LIN {X 0,Y 279.71,Z 650.698,A -85,B 0,C 180,E1 18893.052,E2 18893.052} C_VEL
LIN {X 0,Y 279.473,Z 647.41,A -85,B 0,C 180,E1 18896.902,E2 18896.902} C_VEL
LIN {X 0,Y 279.75,Z 647.577,A -85,B 0,C 180,E1 18903.089,E2 18903.089} C_VEL
LIN {X 0,Y 281.999,Z 655.241,A -85,B 0,C 180,E1 18910.89,E2 18910.89} C_VEL
LIN {X 0,Y 286.328,Z 667.268,A -85,B 0,C 180,E1 18917.884,E2 18917.884} C_VEL
LIN {X 0,Y 291.188,Z 684.37,A -85,B 0,C 180,E1 18924.489,E2 18924.489} C_VEL
LIN {X 0,Y 294.308,Z 701.563,A -85,B 0,C 180,E1 18929.526,E2 18929.526} C_VEL
LIN {X 0,Y 294.245,Z 706.547,A -85,B 0,C 180,E1 18930.593,E2 18930.593} C_VEL
LIN {X 0,Y 277.927,Z 740.652,A -85,B 0,C 180,E1 18934.449,E2 18934.449} C_VEL
LIN {X 0,Y 260.322,Z 771.594,A -85,B 0,C 180,E1 18939.724,E2 18939.724} C_VEL
LIN {X 0,Y 242.682,Z 798.964,A -85,B 0,C 180,E1 18946.842,E2 18946.842} C_VEL
LIN {X 0,Y 228.545,Z 820.039,A -85,B 0,C 180,E1 18955.34,E2 18955.34} C_VEL
LIN {X 0,Y 219.447,Z 834.564,A -85,B 0,C 180,E1 18964.163,E2 18964.163} C_VEL
LIN {X 0,Y 214.489,Z 844.444,A -85,B 0,C 180,E1 18973.653,E2 18973.653} C_VEL
LIN {X 0,Y 212.912,Z 849.596,A -85,B 0,C 180,E1 18982.818,E2 18982.818} C_VEL
LIN {X 0,Y 213.05,Z 850.932,A -85,B 0,C 180,E1 18989.998,E2 18989.998} C_VEL
LIN {X 0,Y 213.023,Z 849.298,A -85,B 0,C 180,E1 18998.143,E2 18998.143} C_VEL
LIN {X 0,Y 215.057,Z 843.186,A -85,B 0,C 180,E1 19007.864,E2 19007.864} C_VEL
LIN {X 0,Y 221.626,Z 830.85,A -85,B 0,C 180,E1 19018.463,E2 19018.463} C_VEL
LIN {X 0,Y 233.239,Z 812.967,A -85,B 0,C 180,E1 19027.923,E2 19027.923} C_VEL
LIN {X 0,Y 248.433,Z 790.316,A -85,B 0,C 180,E1 19035.767,E2 19035.767} C_VEL
LIN {X 0,Y 266.81,Z 760.833,A -85,B 0,C 180,E1 19042.352,E2 19042.352} C_VEL
LIN {X 0,Y 283.537,Z 729.753,A -85,B 0,C 180,E1 19046.951,E2 19046.951} C_VEL
LIN {X 0,Y 294.778,Z 704.676,A -85,B 0,C 180,E1 19049.641,E2 19049.641} C_VEL
LIN {X 0,Y 291.411,Z 685.648,A -85,B 0,C 180,E1 19055.123,E2 19055.123} C_VEL
LIN {X 0,Y 286.674,Z 668.443,A -85,B 0,C 180,E1 19061.593,E2 19061.593} C_VEL
LIN {X 0,Y 282.271,Z 656.335,A -85,B 0,C 180,E1 19068.437,E2 19068.437} C_VEL
LIN {X 0,Y 279.745,Z 647.591,A -85,B 0,C 180,E1 19076.911,E2 19076.911} C_VEL
LIN {X 0,Y 279.623,Z 648.198,A -85,B 0,C 180,E1 19084.646,E2 19084.646} C_VEL
LIN {X 0,Y 282.116,Z 657.702,A -85,B 0,C 180,E1 19093.333,E2 19093.333} C_VEL
LIN {X 0,Y 284.286,Z 663.444,A -85,B 0,C 180,E1 19096.986,E2 19096.986} C_VEL
LIN {X 0,Y 285.392,Z 671.54,A -85,B 0,C 180,E1 19100.105,E2 19100.105} C_VEL
LIN {X 0,Y 286.571,Z 678.848,A -85,B 0,C 180,E1 19102.801,E2 19102.801} C_VEL
LIN {X 0,Y 287.06,Z 679.466,A -85,B 0,C 180,E1 19103.209,E2 19103.209} C_VEL
LIN {X 0,Y 296.62,Z 688.965,A -85,B 0,C 180,E1 19110.583,E2 19110.583} C_VEL
LIN {X 0,Y 304.92,Z 697.051,A -85,B 0,C 180,E1 19117.646,E2 19117.646} C_VEL
LIN {X 0,Y 310.971,Z 702.902,A -85,B 0,C 180,E1 19123.292,E2 19123.292} C_VEL
LIN {X 0,Y 317.433,Z 707.926,A -85,B 0,C 180,E1 19129.521,E2 19129.521} C_VEL
LIN {X 0,Y 322.526,Z 713.626,A -85,B 0,C 180,E1 19135.846,E2 19135.846} C_VEL
LIN {X 0,Y 328,Z 717.173,A -85,B 0,C 180,E1 19142.61,E2 19142.61} C_VEL
LIN {X 0,Y 331.079,Z 721.22,A -85,B 0,C 180,E1 19148.617,E2 19148.617} C_VEL
LIN {X 0,Y 333.856,Z 723.286,A -85,B 0,C 180,E1 19154.266,E2 19154.266} C_VEL
LIN {X 0,Y 336.214,Z 724.311,A -85,B 0,C 180,E1 19160.911,E2 19160.911} C_VEL
LIN {X 0,Y 337.443,Z 724.686,A -85,B 0,C 180,E1 19167.438,E2 19167.438} C_VEL
LIN {X 0,Y 337.436,Z 724.65,A -85,B 0,C 180,E1 19172.564,E2 19172.564} C_VEL
LIN {X 0,Y 336.199,Z 724.407,A -85,B 0,C 180,E1 19179.073,E2 19179.073} C_VEL
LIN {X 0,Y 333.833,Z 723.34,A -85,B 0,C 180,E1 19185.738,E2 19185.738} C_VEL
LIN {X 0,Y 331.067,Z 721.202,A -85,B 0,C 180,E1 19191.387,E2 19191.387} C_VEL
LIN {X 0,Y 327.984,Z 717.14,A -85,B 0,C 180,E1 19197.394,E2 19197.394} C_VEL
LIN {X 0,Y 322.464,Z 713.679,A -85,B 0,C 180,E1 19204.165,E2 19204.165} C_VEL
LIN {X 0,Y 317.373,Z 708.007,A -85,B 0,C 180,E1 19210.466,E2 19210.466} C_VEL
LIN {X 0,Y 310.615,Z 702.32,A -85,B 0,C 180,E1 19217.142,E2 19217.142} C_VEL
LIN {X 0,Y 304.91,Z 697.046,A -85,B 0,C 180,E1 19222.36,E2 19222.36} C_VEL
LIN {X 0,Y 296.59,Z 689.035,A -85,B 0,C 180,E1 19229.414,E2 19229.414} C_VEL
LIN {X 0,Y 287.064,Z 679.509,A -85,B 0,C 180,E1 19236.778,E2 19236.778} C_VEL
LIN {X 0,Y 277.455,Z 660.263,A -85,B 0,C 180,E1 19250.606,E2 19250.606} C_VEL
LIN {X 0,Y 276.701,Z 654.851,A -85,B 0,C 180,E1 19256.871,E2 19256.871} C_VEL
LIN {X 0,Y 276.958,Z 655.076,A -85,B 0,C 180,E1 19263.12,E2 19263.12} C_VEL
LIN {X 0,Y 279.068,Z 662.883,A -85,B 0,C 180,E1 19271.006,E2 19271.006} C_VEL
LIN {X 0,Y 282.954,Z 675.27,A -85,B 0,C 180,E1 19278.105,E2 19278.105} C_VEL
LIN {X 0,Y 286.969,Z 691.731,A -85,B 0,C 180,E1 19284.459,E2 19284.459} C_VEL
LIN {X 0,Y 289.199,Z 707.601,A -85,B 0,C 180,E1 19289.177,E2 19289.177} C_VEL
LIN {X 0,Y 285.282,Z 717.102,A -85,B 0,C 180,E1 19290.276,E2 19290.276} C_VEL
LIN {X 0,Y 268.829,Z 748.728,A -85,B 0,C 180,E1 19294.252,E2 19294.252} C_VEL
LIN {X 0,Y 249.642,Z 780.01,A -85,B 0,C 180,E1 19300.256,E2 19300.256} C_VEL
LIN {X 0,Y 232.045,Z 805.376,A -85,B 0,C 180,E1 19307.849,E2 19307.849} C_VEL
LIN {X 0,Y 218.763,Z 824.231,A -85,B 0,C 180,E1 19316.505,E2 19316.505} C_VEL
LIN {X 0,Y 209.653,Z 838.359,A -85,B 0,C 180,E1 19326.678,E2 19326.678} C_VEL
LIN {X 0,Y 205.697,Z 847.028,A -85,B 0,C 180,E1 19337.284,E2 19337.284} C_VEL
LIN {X 0,Y 204.932,Z 850.268,A -85,B 0,C 180,E1 19345.775,E2 19345.775} C_VEL
LIN {X 0,Y 205.148,Z 850.687,A -85,B 0,C 180,E1 19349.998,E2 19349.998} C_VEL
LIN {X 0,Y 205.128,Z 849.05,A -85,B 0,C 180,E1 19358.459,E2 19358.459} C_VEL
LIN {X 0,Y 207.597,Z 842.427,A -85,B 0,C 180,E1 19369.114,E2 19369.114} C_VEL
LIN {X 0,Y 215.505,Z 829.154,A -85,B 0,C 180,E1 19380.506,E2 19380.506} C_VEL
LIN {X 0,Y 229.199,Z 809.498,A -85,B 0,C 180,E1 19390.551,E2 19390.551} C_VEL
LIN {X 0,Y 245.466,Z 786.097,A -85,B 0,C 180,E1 19398.19,E2 19398.19} C_VEL
LIN {X 0,Y 262.927,Z 758.998,A -85,B 0,C 180,E1 19404.049,E2 19404.049} C_VEL
LIN {X 0,Y 280.537,Z 726.908,A -85,B 0,C 180,E1 19408.637,E2 19408.637} C_VEL
LIN {X 0,Y 289.269,Z 707.475,A -85,B 0,C 180,E1 19410.83,E2 19410.83} C_VEL
LIN {X 0,Y 286.395,Z 689.538,A -85,B 0,C 180,E1 19416.316,E2 19416.316} C_VEL
LIN {X 0,Y 282.277,Z 673.086,A -85,B 0,C 180,E1 19422.932,E2 19422.932} C_VEL
LIN {X 0,Y 278.966,Z 662.903,A -85,B 0,C 180,E1 19429.087,E2 19429.087} C_VEL
LIN {X 0,Y 276.948,Z 655.104,A -85,B 0,C 180,E1 19436.88,E2 19436.88} C_VEL
LIN {X 0,Y 276.7,Z 654.855,A -85,B 0,C 180,E1 19443.129,E2 19443.129} C_VEL
LIN {X 0,Y 278.24,Z 663.042,A -85,B 0,C 180,E1 19451.738,E2 19451.738} C_VEL
LIN {X 0,Y 287.06,Z 679.466,A -85,B 0,C 180,E1 19463.209,E2 19463.209} C_VEL
LIN {X 0,Y 289.006,Z 684.819,A -85,B 0,C 180,E1 19465.563,E2 19465.563} C_VEL
LIN {X 0,Y 290.681,Z 693.974,A -85,B 0,C 180,E1 19469.032,E2 19469.032} C_VEL
LIN {X 0,Y 291.141,Z 694.55,A -85,B 0,C 180,E1 19469.439,E2 19469.439} C_VEL
LIN {X 0,Y 298.491,Z 701.701,A -85,B 0,C 180,E1 19475.552,E2 19475.552} C_VEL
LIN {X 0,Y 306.17,Z 708.716,A -85,B 0,C 180,E1 19482.33,E2 19482.33} C_VEL
LIN {X 0,Y 312.801,Z 714.233,A -85,B 0,C 180,E1 19488.698,E2 19488.698} C_VEL
LIN {X 0,Y 318.348,Z 720.203,A -85,B 0,C 180,E1 19495.334,E2 19495.334} C_VEL
LIN {X 0,Y 324.017,Z 723.954,A -85,B 0,C 180,E1 19502.245,E2 19502.245} C_VEL
LIN {X 0,Y 327.263,Z 728.048,A -85,B 0,C 180,E1 19508.355,E2 19508.355} C_VEL
LIN {X 0,Y 330.039,Z 730.171,A -85,B 0,C 180,E1 19514.079,E2 19514.079} C_VEL
LIN {X 0,Y 332.214,Z 731.196,A -85,B 0,C 180,E1 19519.533,E2 19519.533} C_VEL
LIN {X 0,Y 333.565,Z 731.668,A -85,B 0,C 180,E1 19524.81,E2 19524.81} C_VEL
LIN {X 0,Y 333.984,Z 731.746,A -85,B 0,C 180,E1 19530.001,E2 19530.001} C_VEL
LIN {X 0,Y 333.504,Z 731.607,A -85,B 0,C 180,E1 19535.457,E2 19535.457} C_VEL
LIN {X 0,Y 332.177,Z 731.23,A -85,B 0,C 180,E1 19540.471,E2 19540.471} C_VEL
LIN {X 0,Y 329.918,Z 730.177,A -85,B 0,C 180,E1 19546.148,E2 19546.148} C_VEL
LIN {X 0,Y 326.803,Z 727.575,A -85,B 0,C 180,E1 19552.552,E2 19552.552} C_VEL
LIN {X 0,Y 323.994,Z 723.925,A -85,B 0,C 180,E1 19557.76,E2 19557.76} C_VEL
LIN {X 0,Y 318.253,Z 720.254,A -85,B 0,C 180,E1 19564.681,E2 19564.681} C_VEL
LIN {X 0,Y 312.741,Z 714.248,A -85,B 0,C 180,E1 19571.312,E2 19571.312} C_VEL
LIN {X 0,Y 306.224,Z 708.608,A -85,B 0,C 180,E1 19577.663,E2 19577.663} C_VEL
LIN {X 0,Y 298.52,Z 701.773,A -85,B 0,C 180,E1 19584.452,E2 19584.452} C_VEL
LIN {X 0,Y 291.16,Z 694.683,A -85,B 0,C 180,E1 19590.499,E2 19590.499} C_VEL
LIN {X 0,Y 281.686,Z 684.961,A -85,B 0,C 180,E1 19597.973,E2 19597.973} C_VEL
LIN {X 0,Y 274.243,Z 667.731,A -85,B 0,C 180,E1 19610.495,E2 19610.495} C_VEL
LIN {X 0,Y 273.736,Z 662.251,A -85,B 0,C 180,E1 19616.837,E2 19616.837} C_VEL
LIN {X 0,Y 274.013,Z 662.514,A -85,B 0,C 180,E1 19623.154,E2 19623.154} C_VEL
LIN {X 0,Y 276.148,Z 671.4,A -85,B 0,C 180,E1 19631.872,E2 19631.872} C_VEL
LIN {X 0,Y 279.578,Z 684.378,A -85,B 0,C 180,E1 19638.892,E2 19638.892} C_VEL
LIN {X 0,Y 282.794,Z 701.417,A -85,B 0,C 180,E1 19645.266,E2 19645.266} C_VEL
LIN {X 0,Y 283.599,Z 712.093,A -85,B 0,C 180,E1 19648.403,E2 19648.403} C_VEL
LIN {X 0,Y 266.136,Z 745.555,A -85,B 0,C 180,E1 19652.362,E2 19652.362} C_VEL
LIN {X 0,Y 246.652,Z 776.392,A -85,B 0,C 180,E1 19658.027,E2 19658.027} C_VEL
LIN {X 0,Y 229.143,Z 800.952,A -85,B 0,C 180,E1 19664.93,E2 19664.93} C_VEL
LIN {X 0,Y 213.714,Z 821.702,A -85,B 0,C 180,E1 19673.996,E2 19673.996} C_VEL
LIN {X 0,Y 202.951,Z 836.931,A -85,B 0,C 180,E1 19684.687,E2 19684.687} C_VEL
LIN {X 0,Y 198.392,Z 845.425,A -85,B 0,C 180,E1 19694.559,E2 19694.559} C_VEL
LIN {X 0,Y 197.013,Z 849.79,A -85,B 0,C 180,E1 19704.643,E2 19704.643} C_VEL
LIN {X 0,Y 197.242,Z 850.441,A -85,B 0,C 180,E1 19709.998,E2 19709.998} C_VEL
LIN {X 0,Y 197.256,Z 848.803,A -85,B 0,C 180,E1 19718.799,E2 19718.799} C_VEL
LIN {X 0,Y 199.955,Z 842.175,A -85,B 0,C 180,E1 19729.874,E2 19729.874} C_VEL
LIN {X 0,Y 208.496,Z 828.9,A -85,B 0,C 180,E1 19741.648,E2 19741.648} C_VEL
LIN {X 0,Y 222.947,Z 809.328,A -85,B 0,C 180,E1 19751.888,E2 19751.888} C_VEL
LIN {X 0,Y 240.104,Z 785.844,A -85,B 0,C 180,E1 19759.641,E2 19759.641} C_VEL
LIN {X 0,Y 259.035,Z 757.488,A -85,B 0,C 180,E1 19765.73,E2 19765.73} C_VEL
LIN {X 0,Y 278.307,Z 722.98,A -85,B 0,C 180,E1 19770.497,E2 19770.497} C_VEL
LIN {X 0,Y 283.598,Z 711.983,A -85,B 0,C 180,E1 19771.627,E2 19771.627} C_VEL
LIN {X 0,Y 282.006,Z 696.759,A -85,B 0,C 180,E1 19776.341,E2 19776.341} C_VEL
LIN {X 0,Y 278.752,Z 681.007,A -85,B 0,C 180,E1 19782.682,E2 19782.682} C_VEL
LIN {X 0,Y 275.728,Z 670.419,A -85,B 0,C 180,E1 19788.957,E2 19788.957} C_VEL
LIN {X 0,Y 273.996,Z 662.558,A -85,B 0,C 180,E1 19796.846,E2 19796.846} C_VEL
LIN {X 0,Y 273.741,Z 662.238,A -85,B 0,C 180,E1 19803.163,E2 19803.163} C_VEL
LIN {X 0,Y 274.935,Z 670.536,A -85,B 0,C 180,E1 19811.881,E2 19811.881} C_VEL
LIN {X 0,Y 289.287,Z 692.824,A -85,B 0,C 180,E1 19828.003,E2 19828.003} C_VEL
LIN {X 0,Y 291.141,Z 694.55,A -85,B 0,C 180,E1 19829.439,E2 19829.439} C_VEL
LIN {X 0,Y 292.88,Z 699.556,A -85,B 0,C 180,E1 19831.803,E2 19831.803} C_VEL
LIN {X 0,Y 294.139,Z 708.103,A -85,B 0,C 180,E1 19835.31,E2 19835.31} C_VEL
LIN {X 0,Y 294.559,Z 708.63,A -85,B 0,C 180,E1 19835.719,E2 19835.719} C_VEL
LIN {X 0,Y 301.03,Z 714.193,A -85,B 0,C 180,E1 19841.245,E2 19841.245} C_VEL
LIN {X 0,Y 307.376,Z 720.096,A -85,B 0,C 180,E1 19847.429,E2 19847.429} C_VEL
LIN {X 0,Y 312.591,Z 725.293,A -85,B 0,C 180,E1 19853.267,E2 19853.267} C_VEL
LIN {X 0,Y 317.35,Z 729.041,A -85,B 0,C 180,E1 19858.864,E2 19858.864} C_VEL
LIN {X 0,Y 320.665,Z 731.639,A -85,B 0,C 180,E1 19863.4,E2 19863.4} C_VEL
LIN {X 0,Y 323.556,Z 735.147,A -85,B 0,C 180,E1 19868.875,E2 19868.875} C_VEL
LIN {X 0,Y 327.259,Z 737.599,A -85,B 0,C 180,E1 19876.672,E2 19876.672} C_VEL
LIN {X 0,Y 329.125,Z 738.27,A -85,B 0,C 180,E1 19882.095,E2 19882.095} C_VEL
LIN {X 0,Y 329.948,Z 738.567,A -85,B 0,C 180,E1 19887.38,E2 19887.38} C_VEL
LIN {X 0,Y 329.944,Z 738.537,A -85,B 0,C 180,E1 19892.623,E2 19892.623} C_VEL
LIN {X 0,Y 328.996,Z 738.369,A -85,B 0,C 180,E1 19897.91,E2 19897.91} C_VEL
LIN {X 0,Y 326.862,Z 737.475,A -85,B 0,C 180,E1 19904.18,E2 19904.18} C_VEL
LIN {X 0,Y 323.55,Z 735.142,A -85,B 0,C 180,E1 19911.122,E2 19911.122} C_VEL
LIN {X 0,Y 319.688,Z 730.559,A -85,B 0,C 180,E1 19918.167,E2 19918.167} C_VEL
LIN {X 0,Y 313.763,Z 726.596,A -85,B 0,C 180,E1 19925.25,E2 19925.25} C_VEL
LIN {X 0,Y 309.302,Z 721.596,A -85,B 0,C 180,E1 19930.689,E2 19930.689} C_VEL
LIN {X 0,Y 302.704,Z 716.09,A -85,B 0,C 180,E1 19937.052,E2 19937.052} C_VEL
LIN {X 0,Y 295.761,Z 709.731,A -85,B 0,C 180,E1 19943.281,E2 19943.281} C_VEL
LIN {X 0,Y 287.549,Z 701.861,A -85,B 0,C 180,E1 19950.093,E2 19950.093} C_VEL
LIN {X 0,Y 277.969,Z 692.104,A -85,B 0,C 180,E1 19957.663,E2 19957.663} C_VEL
LIN {X 0,Y 270.876,Z 675.179,A -85,B 0,C 180,E1 19970.376,E2 19970.376} C_VEL
LIN {X 0,Y 270.494,Z 669.57,A -85,B 0,C 180,E1 19976.799,E2 19976.799} C_VEL
LIN {X 0,Y 270.786,Z 669.853,A -85,B 0,C 180,E1 19983.191,E2 19983.191} C_VEL
LIN {X 0,Y 272.7,Z 678.907,A -85,B 0,C 180,E1 19991.973,E2 19991.973} C_VEL
LIN {X 0,Y 275.351,Z 690.526,A -85,B 0,C 180,E1 19998.364,E2 19998.364} C_VEL
LIN {X 0,Y 277.785,Z 706.246,A -85,B 0,C 180,E1 20004.467,E2 20004.467} C_VEL
LIN {X 0,Y 278.057,Z 715.532,A -85,B 0,C 180,E1 20007.307,E2 20007.307} C_VEL
LIN {X 0,Y 260.285,Z 747.905,A -85,B 0,C 180,E1 20011.26,E2 20011.26} C_VEL
LIN {X 0,Y 239.434,Z 779.504,A -85,B 0,C 180,E1 20017.278,E2 20017.278} C_VEL
LIN {X 0,Y 219.66,Z 805.536,A -85,B 0,C 180,E1 20025.237,E2 20025.237} C_VEL
LIN {X 0,Y 205.334,Z 823.723,A -85,B 0,C 180,E1 20033.988,E2 20033.988} C_VEL
LIN {X 0,Y 194.126,Z 839.03,A -85,B 0,C 180,E1 20045.912,E2 20045.912} C_VEL
LIN {X 0,Y 190.059,Z 846.529,A -85,B 0,C 180,E1 20056.218,E2 20056.218} C_VEL
LIN {X 0,Y 189.135,Z 849.776,A -85,B 0,C 180,E1 20065.422,E2 20065.422} C_VEL
LIN {X 0,Y 189.344,Z 850.196,A -85,B 0,C 180,E1 20069.998,E2 20069.998} C_VEL
LIN {X 0,Y 189.376,Z 848.555,A -85,B 0,C 180,E1 20079.168,E2 20079.168} C_VEL
LIN {X 0,Y 192.459,Z 841.764,A -85,B 0,C 180,E1 20090.883,E2 20090.883} C_VEL
LIN {X 0,Y 201.584,Z 828.646,A -85,B 0,C 180,E1 20102.866,E2 20102.866} C_VEL
LIN {X 0,Y 216.45,Z 809.655,A -85,B 0,C 180,E1 20113.078,E2 20113.078} C_VEL
LIN {X 0,Y 233.805,Z 787.105,A -85,B 0,C 180,E1 20120.757,E2 20120.757} C_VEL
LIN {X 0,Y 254.194,Z 757.797,A -85,B 0,C 180,E1 20127.146,E2 20127.146} C_VEL
LIN {X 0,Y 273.847,Z 723.813,A -85,B 0,C 180,E1 20131.841,E2 20131.841} C_VEL
LIN {X 0,Y 278.298,Z 714.952,A -85,B 0,C 180,E1 20132.765,E2 20132.765} C_VEL
LIN {X 0,Y 276.589,Z 698.401,A -85,B 0,C 180,E1 20138.394,E2 20138.394} C_VEL
LIN {X 0,Y 273.88,Z 684.149,A -85,B 0,C 180,E1 20144.832,E2 20144.832} C_VEL
LIN {X 0,Y 271.835,Z 675.929,A -85,B 0,C 180,E1 20150.417,E2 20150.417} C_VEL
LIN {X 0,Y 270.759,Z 669.915,A -85,B 0,C 180,E1 20156.809,E2 20156.809} C_VEL
LIN {X 0,Y 270.513,Z 669.528,A -85,B 0,C 180,E1 20163.201,E2 20163.201} C_VEL
LIN {X 0,Y 271.453,Z 677.943,A -85,B 0,C 180,E1 20172.036,E2 20172.036} C_VEL
LIN {X 0,Y 285.601,Z 700.022,A -85,B 0,C 180,E1 20188.397,E2 20188.397} C_VEL
LIN {X 0,Y 293.249,Z 707.25,A -85,B 0,C 180,E1 20194.583,E2 20194.583} C_VEL
LIN {X 0,Y 294.559,Z 708.63,A -85,B 0,C 180,E1 20195.719,E2 20195.719} C_VEL
LIN {X 0,Y 296.205,Z 715.095,A -85,B 0,C 180,E1 20198.864,E2 20198.864} C_VEL
LIN {X 0,Y 297.369,Z 721.704,A -85,B 0,C 180,E1 20202.024,E2 20202.024} C_VEL
LIN {X 0,Y 303.814,Z 727.288,A -85,B 0,C 180,E1 20208.165,E2 20208.165} C_VEL
LIN {X 0,Y 309.045,Z 732.649,A -85,B 0,C 180,E1 20214.132,E2 20214.132} C_VEL
LIN {X 0,Y 315.127,Z 737.053,A -85,B 0,C 180,E1 20221.391,E2 20221.391} C_VEL
LIN {X 0,Y 318.706,Z 741.187,A -85,B 0,C 180,E1 20227.743,E2 20227.743} C_VEL
LIN {X 0,Y 321.732,Z 743.632,A -85,B 0,C 180,E1 20233.657,E2 20233.657} C_VEL
LIN {X 0,Y 324.049,Z 744.718,A -85,B 0,C 180,E1 20239.266,E2 20239.266} C_VEL
LIN {X 0,Y 325.445,Z 745.215,A -85,B 0,C 180,E1 20244.68,E2 20244.68} C_VEL
LIN {X 0,Y 325.93,Z 745.313,A -85,B 0,C 180,E1 20250.001,E2 20250.001} C_VEL
LIN {X 0,Y 325.449,Z 745.147,A -85,B 0,C 180,E1 20255.322,E2 20255.322} C_VEL
LIN {X 0,Y 323.65,Z 744.628,A -85,B 0,C 180,E1 20261.72,E2 20261.72} C_VEL
LIN {X 0,Y 321.762,Z 743.668,A -85,B 0,C 180,E1 20266.345,E2 20266.345} C_VEL
LIN {X 0,Y 318.694,Z 741.179,A -85,B 0,C 180,E1 20272.261,E2 20272.261} C_VEL
LIN {X 0,Y 315.101,Z 737.015,A -85,B 0,C 180,E1 20278.615,E2 20278.615} C_VEL
LIN {X 0,Y 308.934,Z 732.7,A -85,B 0,C 180,E1 20285.886,E2 20285.886} C_VEL
LIN {X 0,Y 303.804,Z 727.324,A -85,B 0,C 180,E1 20291.832,E2 20291.832} C_VEL
LIN {X 0,Y 296.81,Z 720.849,A -85,B 0,C 180,E1 20298.626,E2 20298.626} C_VEL
LIN {X 0,Y 289.338,Z 714.402,A -85,B 0,C 180,E1 20304.989,E2 20304.989} C_VEL
LIN {X 0,Y 281.693,Z 707.153,A -85,B 0,C 180,E1 20311.173,E2 20311.173} C_VEL
LIN {X 0,Y 267.217,Z 682.501,A -85,B 0,C 180,E1 20330.243,E2 20330.243} C_VEL
LIN {X 0,Y 267.118,Z 676.848,A -85,B 0,C 180,E1 20336.758,E2 20336.758} C_VEL
LIN {X 0,Y 267.443,Z 677.132,A -85,B 0,C 180,E1 20343.231,E2 20343.231} C_VEL
LIN {X 0,Y 268.765,Z 685.164,A -85,B 0,C 180,E1 20351.329,E2 20351.329} C_VEL
LIN {X 0,Y 270.925,Z 696.534,A -85,B 0,C 180,E1 20357.837,E2 20357.837} C_VEL
LIN {X 0,Y 272.703,Z 712.128,A -85,B 0,C 180,E1 20364.081,E2 20364.081} C_VEL
LIN {X 0,Y 272.952,Z 718.045,A -85,B 0,C 180,E1 20366.025,E2 20366.025} C_VEL
LIN {X 0,Y 254.509,Z 750.272,A -85,B 0,C 180,E1 20370.124,E2 20370.124} C_VEL
LIN {X 0,Y 233.714,Z 780.387,A -85,B 0,C 180,E1 20375.98,E2 20375.98} C_VEL
LIN {X 0,Y 212.984,Z 806.491,A -85,B 0,C 180,E1 20384.16,E2 20384.16} C_VEL
LIN {X 0,Y 197.301,Z 825.174,A -85,B 0,C 180,E1 20393.701,E2 20393.701} C_VEL
LIN {X 0,Y 186.73,Z 838.778,A -85,B 0,C 180,E1 20404.894,E2 20404.894} C_VEL
LIN {X 0,Y 182.277,Z 846.28,A -85,B 0,C 180,E1 20415.617,E2 20415.617} C_VEL
LIN {X 0,Y 181.239,Z 849.53,A -85,B 0,C 180,E1 20425.222,E2 20425.222} C_VEL
LIN {X 0,Y 181.205,Z 849.757,A -85,B 0,C 180,E1 20432.274,E2 20432.274} C_VEL
LIN {X 0,Y 181.818,Z 847.34,A -85,B 0,C 180,E1 20441.973,E2 20441.973} C_VEL
LIN {X 0,Y 186.059,Z 839.778,A -85,B 0,C 180,E1 20453.921,E2 20453.921} C_VEL
LIN {X 0,Y 195.871,Z 826.914,A -85,B 0,C 180,E1 20465.16,E2 20465.16} C_VEL
LIN {X 0,Y 212.023,Z 807.661,A -85,B 0,C 180,E1 20475.372,E2 20475.372} C_VEL
LIN {X 0,Y 231.715,Z 782.984,A -85,B 0,C 180,E1 20483.345,E2 20483.345} C_VEL
LIN {X 0,Y 251.613,Z 754.793,A -85,B 0,C 180,E1 20489.166,E2 20489.166} C_VEL
LIN {X 0,Y 271.528,Z 721.107,A -85,B 0,C 180,E1 20493.607,E2 20493.607} C_VEL
LIN {X 0,Y 272.917,Z 717.374,A -85,B 0,C 180,E1 20494.192,E2 20494.192} C_VEL
LIN {X 0,Y 271.558,Z 701.542,A -85,B 0,C 180,E1 20499.999,E2 20499.999} C_VEL
LIN {X 0,Y 269.535,Z 689.194,A -85,B 0,C 180,E1 20506.117,E2 20506.117} C_VEL
LIN {X 0,Y 267.815,Z 681.521,A -85,B 0,C 180,E1 20511.906,E2 20511.906} C_VEL
LIN {X 0,Y 267.402,Z 677.215,A -85,B 0,C 180,E1 20516.768,E2 20516.768} C_VEL
LIN {X 0,Y 267.147,Z 676.79,A -85,B 0,C 180,E1 20523.241,E2 20523.241} C_VEL
LIN {X 0,Y 267.783,Z 685.334,A -85,B 0,C 180,E1 20532.203,E2 20532.203} C_VEL
LIN {X 0,Y 281.7,Z 707.053,A -85,B 0,C 180,E1 20548.827,E2 20548.827} C_VEL
LIN {X 0,Y 289.371,Z 714.363,A -85,B 0,C 180,E1 20555.007,E2 20555.007} C_VEL
LIN {X 0,Y 297.369,Z 721.704,A -85,B 0,C 180,E1 20562.024,E2 20562.024} C_VEL
LIN {X 0,Y 298.37,Z 728.09,A -85,B 0,C 180,E1 20565.156,E2 20565.156} C_VEL
LIN {X 0,Y 299.408,Z 733.898,A -85,B 0,C 180,E1 20568.318,E2 20568.318} C_VEL
LIN {X 0,Y 305.293,Z 739.854,A -85,B 0,C 180,E1 20575.097,E2 20575.097} C_VEL
LIN {X 0,Y 311.433,Z 744.284,A -85,B 0,C 180,E1 20582.494,E2 20582.494} C_VEL
LIN {X 0,Y 314.039,Z 747.504,A -85,B 0,C 180,E1 20587.394,E2 20587.394} C_VEL
LIN {X 0,Y 317.107,Z 750.049,A -85,B 0,C 180,E1 20593.411,E2 20593.411} C_VEL
LIN {X 0,Y 319.593,Z 751.233,A -85,B 0,C 180,E1 20599.115,E2 20599.115} C_VEL
LIN {X 0,Y 321.084,Z 751.797,A -85,B 0,C 180,E1 20604.608,E2 20604.608} C_VEL
LIN {X 0,Y 321.585,Z 751.874,A -85,B 0,C 180,E1 20610.001,E2 20610.001} C_VEL
LIN {X 0,Y 321.084,Z 751.737,A -85,B 0,C 180,E1 20615.395,E2 20615.395} C_VEL
LIN {X 0,Y 319.488,Z 751.274,A -85,B 0,C 180,E1 20620.892,E2 20620.892} C_VEL
LIN {X 0,Y 316.599,Z 749.777,A -85,B 0,C 180,E1 20627.58,E2 20627.58} C_VEL
LIN {X 0,Y 313.438,Z 746.779,A -85,B 0,C 180,E1 20633.827,E2 20633.827} C_VEL
LIN {X 0,Y 310.237,Z 743.293,A -85,B 0,C 180,E1 20639.106,E2 20639.106} C_VEL
LIN {X 0,Y 305.219,Z 739.92,A -85,B 0,C 180,E1 20644.888,E2 20644.888} C_VEL
LIN {X 0,Y 298.885,Z 733.47,A -85,B 0,C 180,E1 20652.213,E2 20652.213} C_VEL
LIN {X 0,Y 291.366,Z 726.507,A -85,B 0,C 180,E1 20659.409,E2 20659.409} C_VEL
LIN {X 0,Y 282.523,Z 718.493,A -85,B 0,C 180,E1 20666.876,E2 20666.876} C_VEL
LIN {X 0,Y 272.743,Z 709.022,A -85,B 0,C 180,E1 20674.606,E2 20674.606} C_VEL
LIN {X 0,Y 263.294,Z 688.458,A -85,B 0,C 180,E1 20691.388,E2 20691.388} C_VEL
LIN {X 0,Y 263.482,Z 684.023,A -85,B 0,C 180,E1 20696.713,E2 20696.713} C_VEL
LIN {X 0,Y 263.604,Z 683.395,A -85,B 0,C 180,E1 20699.997,E2 20699.997} C_VEL
LIN {X 0,Y 263.761,Z 685.688,A -85,B 0,C 180,E1 20704.919,E2 20704.919} C_VEL
LIN {X 0,Y 264.959,Z 692.557,A -85,B 0,C 180,E1 20711.494,E2 20711.494} C_VEL
LIN {X 0,Y 266.63,Z 704.336,A -85,B 0,C 180,E1 20718.134,E2 20718.134} C_VEL
LIN {X 0,Y 267.645,Z 719.467,A -85,B 0,C 180,E1 20724.197,E2 20724.197} C_VEL
LIN {X 0,Y 266.673,Z 723.303,A -85,B 0,C 180,E1 20725.121,E2 20725.121} C_VEL
LIN {X 0,Y 246.257,Z 756.605,A -85,B 0,C 180,E1 20729.568,E2 20729.568} C_VEL
LIN {X 0,Y 224.783,Z 785.425,A -85,B 0,C 180,E1 20735.702,E2 20735.702} C_VEL
LIN {X 0,Y 206.379,Z 807.4,A -85,B 0,C 180,E1 20743.011,E2 20743.011} C_VEL
LIN {X 0,Y 188.667,Z 827.356,A -85,B 0,C 180,E1 20753.888,E2 20753.888} C_VEL
LIN {X 0,Y 178.601,Z 839.52,A -85,B 0,C 180,E1 20765.008,E2 20765.008} C_VEL
LIN {X 0,Y 174.025,Z 847.09,A -85,B 0,C 180,E1 20777.478,E2 20777.478} C_VEL
LIN {X 0,Y 173.326,Z 849.284,A -85,B 0,C 180,E1 20785.003,E2 20785.003} C_VEL
LIN {X 0,Y 173.544,Z 849.705,A -85,B 0,C 180,E1 20789.998,E2 20789.998} C_VEL
LIN {X 0,Y 173.635,Z 848.059,A -85,B 0,C 180,E1 20800.007,E2 20800.007} C_VEL
LIN {X 0,Y 177.285,Z 841.44,A -85,B 0,C 180,E1 20812.519,E2 20812.519} C_VEL
LIN {X 0,Y 187.692,Z 828.563,A -85,B 0,C 180,E1 20825.261,E2 20825.261} C_VEL
LIN {X 0,Y 204.476,Z 809.5,A -85,B 0,C 180,E1 20836.051,E2 20836.051} C_VEL
LIN {X 0,Y 223.863,Z 786.6,A -85,B 0,C 180,E1 20843.985,E2 20843.985} C_VEL
LIN {X 0,Y 245.584,Z 757.54,A -85,B 0,C 180,E1 20850.288,E2 20850.288} C_VEL
LIN {X 0,Y 265.908,Z 724.618,A -85,B 0,C 180,E1 20854.745,E2 20854.745} C_VEL
LIN {X 0,Y 267.419,Z 721.962,A -85,B 0,C 180,E1 20855.03,E2 20855.03} C_VEL
LIN {X 0,Y 266.945,Z 708.191,A -85,B 0,C 180,E1 20860.177,E2 20860.177} C_VEL
LIN {X 0,Y 265.55,Z 696.755,A -85,B 0,C 180,E1 20865.821,E2 20865.821} C_VEL
LIN {X 0,Y 264.16,Z 688.774,A -85,B 0,C 180,E1 20871.793,E2 20871.793} C_VEL
LIN {X 0,Y 263.758,Z 684.402,A -85,B 0,C 180,E1 20876.724,E2 20876.724} C_VEL
LIN {X 0,Y 263.611,Z 683.381,A -85,B 0,C 180,E1 20880.003,E2 20880.003} C_VEL
LIN {X 0,Y 263.289,Z 685.236,A -85,B 0,C 180,E1 20884.935,E2 20884.935} C_VEL
LIN {X 0,Y 263.946,Z 693.811,A -85,B 0,C 180,E1 20893.223,E2 20893.223} C_VEL
LIN {X 0,Y 278.598,Z 714.735,A -85,B 0,C 180,E1 20909.934,E2 20909.934} C_VEL
LIN {X 0,Y 286.487,Z 722.445,A -85,B 0,C 180,E1 20916.497,E2 20916.497} C_VEL
LIN {X 0,Y 293.505,Z 728.991,A -85,B 0,C 180,E1 20922.734,E2 20922.734} C_VEL
LIN {X 0,Y 299.408,Z 733.898,A -85,B 0,C 180,E1 20928.318,E2 20928.318} C_VEL
LIN {X 0,Y 300.171,Z 737.996,A -85,B 0,C 180,E1 20930.697,E2 20930.697} C_VEL
LIN {X 0,Y 299.872,Z 745.37,A -85,B 0,C 180,E1 20934.231,E2 20934.231} C_VEL
LIN {X 0,Y 300.126,Z 745.786,A -85,B 0,C 180,E1 20934.642,E2 20934.642} C_VEL
LIN {X 0,Y 305.126,Z 749.379,A -85,B 0,C 180,E1 20940.361,E2 20940.361} C_VEL
LIN {X 0,Y 309.152,Z 753.647,A -85,B 0,C 180,E1 20947.016,E2 20947.016} C_VEL
LIN {X 0,Y 312.25,Z 756.307,A -85,B 0,C 180,E1 20953.146,E2 20953.146} C_VEL
LIN {X 0,Y 314.896,Z 757.603,A -85,B 0,C 180,E1 20958.95,E2 20958.95} C_VEL
LIN {X 0,Y 316.363,Z 758.124,A -85,B 0,C 180,E1 20964.527,E2 20964.527} C_VEL
LIN {X 0,Y 316.903,Z 758.212,A -85,B 0,C 180,E1 20970.001,E2 20970.001} C_VEL
LIN {X 0,Y 316.355,Z 758.085,A -85,B 0,C 180,E1 20975.476,E2 20975.476} C_VEL
LIN {X 0,Y 314.79,Z 757.631,A -85,B 0,C 180,E1 20981.056,E2 20981.056} C_VEL
LIN {X 0,Y 312.291,Z 756.328,A -85,B 0,C 180,E1 20986.855,E2 20986.855} C_VEL
LIN {X 0,Y 308.527,Z 752.844,A -85,B 0,C 180,E1 20994.231,E2 20994.231} C_VEL
LIN {X 0,Y 305.08,Z 749.381,A -85,B 0,C 180,E1 20999.647,E2 20999.647} C_VEL
LIN {X 0,Y 298.38,Z 744.16,A -85,B 0,C 180,E1 21007.366,E2 21007.366} C_VEL
LIN {X 0,Y 292.411,Z 738.512,A -85,B 0,C 180,E1 21013.737,E2 21013.737} C_VEL
LIN {X 0,Y 285.203,Z 731.626,A -85,B 0,C 180,E1 21020.583,E2 21020.583} C_VEL
LIN {X 0,Y 275.532,Z 722.656,A -85,B 0,C 180,E1 21028.645,E2 21028.645} C_VEL
LIN {X 0,Y 260.996,Z 705.079,A -85,B 0,C 180,E1 21043.193,E2 21043.193} C_VEL
LIN {X 0,Y 259.272,Z 693.76,A -85,B 0,C 180,E1 21053.312,E2 21053.312} C_VEL
LIN {X 0,Y 259.696,Z 691.122,A -85,B 0,C 180,E1 21056.665,E2 21056.665} C_VEL
LIN {X 0,Y 259.934,Z 690.388,A -85,B 0,C 180,E1 21059.997,E2 21059.997} C_VEL
LIN {X 0,Y 259.973,Z 692.782,A -85,B 0,C 180,E1 21064.991,E2 21064.991} C_VEL
LIN {X 0,Y 260.859,Z 699.836,A -85,B 0,C 180,E1 21071.676,E2 21071.676} C_VEL
LIN {X 0,Y 262.005,Z 711.959,A -85,B 0,C 180,E1 21078.464,E2 21078.464} C_VEL
LIN {X 0,Y 262.245,Z 724.998,A -85,B 0,C 180,E1 21083.749,E2 21083.749} C_VEL
LIN {X 0,Y 241.631,Z 757.375,A -85,B 0,C 180,E1 21088.068,E2 21088.068} C_VEL
LIN {X 0,Y 219.177,Z 786.338,A -85,B 0,C 180,E1 21094.288,E2 21094.288} C_VEL
LIN {X 0,Y 199.277,Z 808.815,A -85,B 0,C 180,E1 21102.052,E2 21102.052} C_VEL
LIN {X 0,Y 181.926,Z 827.344,A -85,B 0,C 180,E1 21112.544,E2 21112.544} C_VEL
LIN {X 0,Y 171.279,Z 839.268,A -85,B 0,C 180,E1 21123.861,E2 21123.861} C_VEL
LIN {X 0,Y 166.215,Z 846.842,A -85,B 0,C 180,E1 21136.879,E2 21136.879} C_VEL
LIN {X 0,Y 165.43,Z 849.038,A -85,B 0,C 180,E1 21144.764,E2 21144.764} C_VEL
LIN {X 0,Y 165.635,Z 849.46,A -85,B 0,C 180,E1 21149.998,E2 21149.998} C_VEL
LIN {X 0,Y 165.785,Z 847.811,A -85,B 0,C 180,E1 21160.486,E2 21160.486} C_VEL
LIN {X 0,Y 169.816,Z 841.188,A -85,B 0,C 180,E1 21173.568,E2 21173.568} C_VEL
LIN {X 0,Y 180.083,Z 829.329,A -85,B 0,C 180,E1 21185.911,E2 21185.911} C_VEL
LIN {X 0,Y 196.077,Z 812.292,A -85,B 0,C 180,E1 21196.341,E2 21196.341} C_VEL
LIN {X 0,Y 216.718,Z 789.32,A -85,B 0,C 180,E1 21204.897,E2 21204.897} C_VEL
LIN {X 0,Y 238.796,Z 761.206,A -85,B 0,C 180,E1 21211.255,E2 21211.255} C_VEL
LIN {X 0,Y 259.074,Z 730.531,A -85,B 0,C 180,E1 21215.643,E2 21215.643} C_VEL
LIN {X 0,Y 262.052,Z 725.286,A -85,B 0,C 180,E1 21216.233,E2 21216.233} C_VEL
LIN {X 0,Y 261.933,Z 712.077,A -85,B 0,C 180,E1 21221.531,E2 21221.531} C_VEL
LIN {X 0,Y 260.979,Z 701.137,A -85,B 0,C 180,E1 21227.482,E2 21227.482} C_VEL
LIN {X 0,Y 259.982,Z 694.369,A -85,B 0,C 180,E1 21233.337,E2 21233.337} C_VEL
LIN {X 0,Y 259.996,Z 691.529,A -85,B 0,C 180,E1 21236.676,E2 21236.676} C_VEL
LIN {X 0,Y 259.932,Z 690.392,A -85,B 0,C 180,E1 21240.003,E2 21240.003} C_VEL
LIN {X 0,Y 259.437,Z 692.327,A -85,B 0,C 180,E1 21245.009,E2 21245.009} C_VEL
LIN {X 0,Y 259.676,Z 699.884,A -85,B 0,C 180,E1 21252.59,E2 21252.59} C_VEL
LIN {X 0,Y 273.502,Z 720.751,A -85,B 0,C 180,E1 21269.776,E2 21269.776} C_VEL
LIN {X 0,Y 281.706,Z 728.733,A -85,B 0,C 180,E1 21276.536,E2 21276.536} C_VEL
LIN {X 0,Y 288.948,Z 735.532,A -85,B 0,C 180,E1 21283.02,E2 21283.02} C_VEL
LIN {X 0,Y 296.113,Z 741.511,A -85,B 0,C 180,E1 21289.858,E2 21289.858} C_VEL
LIN {X 0,Y 300.126,Z 745.786,A -85,B 0,C 180,E1 21294.642,E2 21294.642} C_VEL
LIN {X 0,Y 300.462,Z 751.07,A -85,B 0,C 180,E1 21297.832,E2 21297.832} C_VEL
LIN {X 0,Y 300.572,Z 755.928,A -85,B 0,C 180,E1 21301.06,E2 21301.06} C_VEL
LIN {X 0,Y 303.95,Z 759.528,A -85,B 0,C 180,E1 21306.6,E2 21306.6} C_VEL
LIN {X 0,Y 307.186,Z 762.413,A -85,B 0,C 180,E1 21312.859,E2 21312.859} C_VEL
LIN {X 0,Y 309.846,Z 763.731,A -85,B 0,C 180,E1 21318.768,E2 21318.768} C_VEL
LIN {X 0,Y 311.455,Z 764.306,A -85,B 0,C 180,E1 21324.441,E2 21324.441} C_VEL
LIN {X 0,Y 312.04,Z 764.427,A -85,B 0,C 180,E1 21330.001,E2 21330.001} C_VEL
LIN {X 0,Y 311.443,Z 764.276,A -85,B 0,C 180,E1 21335.562,E2 21335.562} C_VEL
LIN {X 0,Y 309.234,Z 763.566,A -85,B 0,C 180,E1 21342.577,E2 21342.577} C_VEL
LIN {X 0,Y 307.225,Z 762.423,A -85,B 0,C 180,E1 21347.141,E2 21347.141} C_VEL
LIN {X 0,Y 303.95,Z 759.492,A -85,B 0,C 180,E1 21353.403,E2 21353.403} C_VEL
LIN {X 0,Y 301.199,Z 756.329,A -85,B 0,C 180,E1 21358.164,E2 21358.164} C_VEL
LIN {X 0,Y 295.289,Z 752.122,A -85,B 0,C 180,E1 21365.146,E2 21365.146} C_VEL
LIN {X 0,Y 290.374,Z 747.069,A -85,B 0,C 180,E1 21370.843,E2 21370.843} C_VEL
LIN {X 0,Y 282.591,Z 739.986,A -85,B 0,C 180,E1 21378.384,E2 21378.384} C_VEL
LIN {X 0,Y 274.029,Z 732.282,A -85,B 0,C 180,E1 21385.694,E2 21385.694} C_VEL
LIN {X 0,Y 264.234,Z 722.958,A -85,B 0,C 180,E1 21393.492,E2 21393.492} C_VEL
LIN {X 0,Y 255.173,Z 702.219,A -85,B 0,C 180,E1 21411.472,E2 21411.472} C_VEL
LIN {X 0,Y 255.709,Z 698.116,A -85,B 0,C 180,E1 21416.613,E2 21416.613} C_VEL
LIN {X 0,Y 256.022,Z 697.263,A -85,B 0,C 180,E1 21419.996,E2 21419.996} C_VEL
LIN {X 0,Y 255.982,Z 699.749,A -85,B 0,C 180,E1 21425.069,E2 21425.069} C_VEL
LIN {X 0,Y 256.619,Z 707.041,A -85,B 0,C 180,E1 21431.873,E2 21431.873} C_VEL
LIN {X 0,Y 257.174,Z 718.745,A -85,B 0,C 180,E1 21438.409,E2 21438.409} C_VEL
LIN {X 0,Y 256.628,Z 728.9,A -85,B 0,C 180,E1 21442.543,E2 21442.543} C_VEL
LIN {X 0,Y 236.458,Z 759.07,A -85,B 0,C 180,E1 21446.687,E2 21446.687} C_VEL
LIN {X 0,Y 213.426,Z 787.602,A -85,B 0,C 180,E1 21452.898,E2 21452.898} C_VEL
LIN {X 0,Y 192.535,Z 809.92,A -85,B 0,C 180,E1 21460.876,E2 21460.876} C_VEL
LIN {X 0,Y 174.831,Z 827.808,A -85,B 0,C 180,E1 21471.442,E2 21471.442} C_VEL
LIN {X 0,Y 162.366,Z 840.931,A -85,B 0,C 180,E1 21485.275,E2 21485.275} C_VEL
LIN {X 0,Y 157.948,Z 847.562,A -85,B 0,C 180,E1 21498.982,E2 21498.982} C_VEL
LIN {X 0,Y 157.726,Z 849.214,A -85,B 0,C 180,E1 21509.997,E2 21509.997} C_VEL
LIN {X 0,Y 157.936,Z 847.563,A -85,B 0,C 180,E1 21521.014,E2 21521.014} C_VEL
LIN {X 0,Y 162.419,Z 840.936,A -85,B 0,C 180,E1 21534.711,E2 21534.711} C_VEL
LIN {X 0,Y 174.784,Z 827.837,A -85,B 0,C 180,E1 21548.54,E2 21548.54} C_VEL
LIN {X 0,Y 194.041,Z 808.39,A -85,B 0,C 180,E1 21559.83,E2 21559.83} C_VEL
LIN {X 0,Y 214.701,Z 786.1,A -85,B 0,C 180,E1 21567.499,E2 21567.499} C_VEL
LIN {X 0,Y 237.875,Z 757.195,A -85,B 0,C 180,E1 21573.642,E2 21573.642} C_VEL
LIN {X 0,Y 256.623,Z 728.94,A -85,B 0,C 180,E1 21577.444,E2 21577.444} C_VEL
LIN {X 0,Y 257.045,Z 716.006,A -85,B 0,C 180,E1 21582.935,E2 21582.935} C_VEL
LIN {X 0,Y 256.493,Z 705.905,A -85,B 0,C 180,E1 21588.981,E2 21588.981} C_VEL
LIN {X 0,Y 256.007,Z 698.515,A -85,B 0,C 180,E1 21596.624,E2 21596.624} C_VEL
LIN {X 0,Y 256.018,Z 697.27,A -85,B 0,C 180,E1 21600.004,E2 21600.004} C_VEL
LIN {X 0,Y 255.43,Z 699.335,A -85,B 0,C 180,E1 21605.087,E2 21605.087} C_VEL
LIN {X 0,Y 255.344,Z 706.994,A -85,B 0,C 180,E1 21612.807,E2 21612.807} C_VEL
LIN {X 0,Y 270.414,Z 728.543,A -85,B 0,C 180,E1 21631.251,E2 21631.251} C_VEL
LIN {X 0,Y 279.008,Z 736.782,A -85,B 0,C 180,E1 21638.464,E2 21638.464} C_VEL
LIN {X 0,Y 286.871,Z 744.206,A -85,B 0,C 180,E1 21645.778,E2 21645.778} C_VEL
LIN {X 0,Y 292.822,Z 749.41,A -85,B 0,C 180,E1 21651.802,E2 21651.802} C_VEL
LIN {X 0,Y 299.615,Z 755.202,A -85,B 0,C 180,E1 21659.76,E2 21659.76} C_VEL
LIN {X 0,Y 300.572,Z 755.928,A -85,B 0,C 180,E1 21661.06,E2 21661.06} C_VEL
LIN {X 0,Y 300.678,Z 759.33,A -85,B 0,C 180,E1 21663.467,E2 21663.467} C_VEL
LIN {X 0,Y 299.217,Z 765.869,A -85,B 0,C 180,E1 21667.377,E2 21667.377} C_VEL
LIN {X 0,Y 299.087,Z 765.932,A -85,B 0,C 180,E1 21667.48,E2 21667.48} C_VEL
LIN {X 0,Y 301.824,Z 768.273,A -85,B 0,C 180,E1 21672.545,E2 21672.545} C_VEL
LIN {X 0,Y 304.608,Z 769.704,A -85,B 0,C 180,E1 21678.572,E2 21678.572} C_VEL
LIN {X 0,Y 306.363,Z 770.33,A -85,B 0,C 180,E1 21684.348,E2 21684.348} C_VEL
LIN {X 0,Y 306.94,Z 770.445,A -85,B 0,C 180,E1 21690.001,E2 21690.001} C_VEL
LIN {X 0,Y 306.346,Z 770.305,A -85,B 0,C 180,E1 21695.655,E2 21695.655} C_VEL
LIN {X 0,Y 304.512,Z 769.707,A -85,B 0,C 180,E1 21701.434,E2 21701.434} C_VEL
LIN {X 0,Y 301.559,Z 768.065,A -85,B 0,C 180,E1 21708.047,E2 21708.047} C_VEL
LIN {X 0,Y 298.21,Z 764.843,A -85,B 0,C 180,E1 21714.373,E2 21714.373} C_VEL
LIN {X 0,Y 294.895,Z 761.537,A -85,B 0,C 180,E1 21719.547,E2 21719.547} C_VEL
LIN {X 0,Y 289.26,Z 757.337,A -85,B 0,C 180,E1 21726.042,E2 21726.042} C_VEL
LIN {X 0,Y 284.02,Z 752.075,A -85,B 0,C 180,E1 21731.938,E2 21731.938} C_VEL
LIN {X 0,Y 276.554,Z 745.14,A -85,B 0,C 180,E1 21739.094,E2 21739.094} C_VEL
LIN {X 0,Y 268.585,Z 737.995,A -85,B 0,C 180,E1 21745.814,E2 21745.814} C_VEL
LIN {X 0,Y 258.552,Z 728.282,A -85,B 0,C 180,E1 21754.037,E2 21754.037} C_VEL
LIN {X 0,Y 250.937,Z 707.609,A -85,B 0,C 180,E1 21773.089,E2 21773.089} C_VEL
LIN {X 0,Y 251.532,Z 704.993,A -85,B 0,C 180,E1 21776.557,E2 21776.557} C_VEL
LIN {X 0,Y 251.957,Z 704.049,A -85,B 0,C 180,E1 21779.996,E2 21779.996} C_VEL
LIN {X 0,Y 251.814,Z 706.632,A -85,B 0,C 180,E1 21785.153,E2 21785.153} C_VEL
LIN {X 0,Y 252.061,Z 712.876,A -85,B 0,C 180,E1 21791.216,E2 21791.216} C_VEL
LIN {X 0,Y 252.086,Z 724.431,A -85,B 0,C 180,E1 21797.942,E2 21797.942} C_VEL
LIN {X 0,Y 251.777,Z 731.479,A -85,B 0,C 180,E1 21801.072,E2 21801.072} C_VEL
LIN {X 0,Y 230.01,Z 762.574,A -85,B 0,C 180,E1 21805.562,E2 21805.562} C_VEL
LIN {X 0,Y 207.793,Z 788.802,A -85,B 0,C 180,E1 21811.424,E2 21811.424} C_VEL
LIN {X 0,Y 183.845,Z 813.078,A -85,B 0,C 180,E1 21820.603,E2 21820.603} C_VEL
LIN {X 0,Y 165.586,Z 830.221,A -85,B 0,C 180,E1 21832.035,E2 21832.035} C_VEL
LIN {X 0,Y 155.052,Z 840.679,A -85,B 0,C 180,E1 21844.024,E2 21844.024} C_VEL
LIN {X 0,Y 150.107,Z 847.314,A -85,B 0,C 180,E1 21858.398,E2 21858.398} C_VEL
LIN {X 0,Y 149.815,Z 848.968,A -85,B 0,C 180,E1 21869.997,E2 21869.997} C_VEL
LIN {X 0,Y 150.097,Z 847.315,A -85,B 0,C 180,E1 21881.597,E2 21881.597} C_VEL
LIN {X 0,Y 155.103,Z 840.685,A -85,B 0,C 180,E1 21895.961,E2 21895.961} C_VEL
LIN {X 0,Y 168.479,Z 827.584,A -85,B 0,C 180,E1 21910.269,E2 21910.269} C_VEL
LIN {X 0,Y 189.194,Z 807.828,A -85,B 0,C 180,E1 21921.868,E2 21921.868} C_VEL
LIN {X 0,Y 211.379,Z 784.798,A -85,B 0,C 180,E1 21929.636,E2 21929.636} C_VEL
LIN {X 0,Y 234.401,Z 756.942,A -85,B 0,C 180,E1 21935.41,E2 21935.41} C_VEL
LIN {X 0,Y 251.77,Z 731.488,A -85,B 0,C 180,E1 21938.928,E2 21938.928} C_VEL
LIN {X 0,Y 252.208,Z 718.344,A -85,B 0,C 180,E1 21945.272,E2 21945.272} C_VEL
LIN {X 0,Y 251.843,Z 709.84,A -85,B 0,C 180,E1 21951.389,E2 21951.389} C_VEL
LIN {X 0,Y 251.854,Z 705.42,A -85,B 0,C 180,E1 21956.569,E2 21956.569} C_VEL
LIN {X 0,Y 251.958,Z 704.047,A -85,B 0,C 180,E1 21960.004,E2 21960.004} C_VEL
LIN {X 0,Y 251.194,Z 706.215,A -85,B 0,C 180,E1 21965.173,E2 21965.173} C_VEL
LIN {X 0,Y 250.928,Z 714.973,A -85,B 0,C 180,E1 21973.922,E2 21973.922} C_VEL
LIN {X 0,Y 265.428,Z 734.705,A -85,B 0,C 180,E1 21991.488,E2 21991.488} C_VEL
LIN {X 0,Y 273.583,Z 742.542,A -85,B 0,C 180,E1 21998.336,E2 21998.336} C_VEL
LIN {X 0,Y 281.768,Z 750.209,A -85,B 0,C 180,E1 22005.878,E2 22005.878} C_VEL
LIN {X 0,Y 287.671,Z 755.406,A -85,B 0,C 180,E1 22011.895,E2 22011.895} C_VEL
LIN {X 0,Y 293.814,Z 760.783,A -85,B 0,C 180,E1 22019.098,E2 22019.098} C_VEL
LIN {X 0,Y 296.674,Z 762.972,A -85,B 0,C 180,E1 22022.758,E2 22022.758} C_VEL
LIN {X 0,Y 299.087,Z 765.932,A -85,B 0,C 180,E1 22027.48,E2 22027.48} C_VEL
LIN {X 0,Y 298.903,Z 768.995,A -85,B 0,C 180,E1 22029.921,E2 22029.921} C_VEL
LIN {X 0,Y 296.985,Z 774.242,A -85,B 0,C 180,E1 22033.571,E2 22033.571} C_VEL
LIN {X 0,Y 297.034,Z 774.441,A -85,B 0,C 180,E1 22033.991,E2 22033.991} C_VEL
LIN {X 0,Y 299.166,Z 775.503,A -85,B 0,C 180,E1 22038.361,E2 22038.361} C_VEL
LIN {X 0,Y 300.937,Z 776.07,A -85,B 0,C 180,E1 22044.246,E2 22044.246} C_VEL
LIN {X 0,Y 301.551,Z 776.223,A -85,B 0,C 180,E1 22050.001,E2 22050.001} C_VEL
LIN {X 0,Y 300.912,Z 776.056,A -85,B 0,C 180,E1 22055.758,E2 22055.758} C_VEL
LIN {X 0,Y 299.074,Z 775.499,A -85,B 0,C 180,E1 22061.645,E2 22061.645} C_VEL
LIN {X 0,Y 296.259,Z 773.884,A -85,B 0,C 180,E1 22067.796,E2 22067.796} C_VEL
LIN {X 0,Y 292.82,Z 770.601,A -85,B 0,C 180,E1 22074.349,E2 22074.349} C_VEL
LIN {X 0,Y 288.909,Z 766.932,A -85,B 0,C 180,E1 22080.222,E2 22080.222} C_VEL
LIN {X 0,Y 282.196,Z 761.285,A -85,B 0,C 180,E1 22088.065,E2 22088.065} C_VEL
LIN {X 0,Y 275.731,Z 755.413,A -85,B 0,C 180,E1 22094.643,E2 22094.643} C_VEL
LIN {X 0,Y 268.02,Z 748.094,A -85,B 0,C 180,E1 22101.73,E2 22101.73} C_VEL
LIN {X 0,Y 259.92,Z 740.465,A -85,B 0,C 180,E1 22108.496,E2 22108.496} C_VEL
LIN {X 0,Y 246.466,Z 714.31,A -85,B 0,C 180,E1 22133.056,E2 22133.056} C_VEL
LIN {X 0,Y 247.17,Z 711.751,A -85,B 0,C 180,E1 22136.496,E2 22136.496} C_VEL
LIN {X 0,Y 247.685,Z 710.716,A -85,B 0,C 180,E1 22139.996,E2 22139.996} C_VEL
LIN {X 0,Y 247.426,Z 713.388,A -85,B 0,C 180,E1 22145.245,E2 22145.245} C_VEL
LIN {X 0,Y 247.408,Z 720.038,A -85,B 0,C 180,E1 22151.535,E2 22151.535} C_VEL
LIN {X 0,Y 246.919,Z 730.776,A -85,B 0,C 180,E1 22157.788,E2 22157.788} C_VEL
LIN {X 0,Y 246.288,Z 735.458,A -85,B 0,C 180,E1 22159.897,E2 22159.897} C_VEL
LIN {X 0,Y 222.978,Z 766.922,A -85,B 0,C 180,E1 22164.533,E2 22164.533} C_VEL
LIN {X 0,Y 198.312,Z 793.986,A -85,B 0,C 180,E1 22171.121,E2 22171.121} C_VEL
LIN {X 0,Y 176.408,Z 814.835,A -85,B 0,C 180,E1 22179.655,E2 22179.655} C_VEL
LIN {X 0,Y 156.138,Z 832.773,A -85,B 0,C 180,E1 22192.837,E2 22192.837} C_VEL
LIN {X 0,Y 144.824,Z 843.539,A -85,B 0,C 180,E1 22208.324,E2 22208.324} C_VEL
LIN {X 0,Y 142.278,Z 847.066,A -85,B 0,C 180,E1 22217.75,E2 22217.75} C_VEL
LIN {X 0,Y 141.903,Z 848.723,A -85,B 0,C 180,E1 22229.997,E2 22229.997} C_VEL
LIN {X 0,Y 142.269,Z 847.066,A -85,B 0,C 180,E1 22242.245,E2 22242.245} C_VEL
LIN {X 0,Y 147.832,Z 840.432,A -85,B 0,C 180,E1 22257.342,E2 22257.342} C_VEL
LIN {X 0,Y 161.791,Z 827.783,A -85,B 0,C 180,E1 22271.751,E2 22271.751} C_VEL
LIN {X 0,Y 182.012,Z 809.613,A -85,B 0,C 180,E1 22282.934,E2 22282.934} C_VEL
LIN {X 0,Y 205.056,Z 787.114,A -85,B 0,C 180,E1 22290.909,E2 22290.909} C_VEL
LIN {X 0,Y 229.626,Z 758.588,A -85,B 0,C 180,E1 22296.925,E2 22296.925} C_VEL
LIN {X 0,Y 246.486,Z 734.816,A -85,B 0,C 180,E1 22300.322,E2 22300.322} C_VEL
LIN {X 0,Y 247.316,Z 722.382,A -85,B 0,C 180,E1 22306.866,E2 22306.866} C_VEL
LIN {X 0,Y 247.315,Z 714.999,A -85,B 0,C 180,E1 22312.994,E2 22312.994} C_VEL
LIN {X 0,Y 247.682,Z 710.72,A -85,B 0,C 180,E1 22320.004,E2 22320.004} C_VEL
LIN {X 0,Y 247.21,Z 711.69,A -85,B 0,C 180,E1 22323.503,E2 22323.503} C_VEL
LIN {X 0,Y 246.074,Z 719.541,A -85,B 0,C 180,E1 22332.218,E2 22332.218} C_VEL
LIN {X 0,Y 260.736,Z 741.147,A -85,B 0,C 180,E1 22352.121,E2 22352.121} C_VEL
LIN {X 0,Y 269.032,Z 749.012,A -85,B 0,C 180,E1 22359.107,E2 22359.107} C_VEL
LIN {X 0,Y 277.301,Z 756.748,A -85,B 0,C 180,E1 22366.838,E2 22366.838} C_VEL
LIN {X 0,Y 283.187,Z 762.187,A -85,B 0,C 180,E1 22373.067,E2 22373.067} C_VEL
LIN {X 0,Y 288.936,Z 766.915,A -85,B 0,C 180,E1 22379.769,E2 22379.769} C_VEL
LIN {X 0,Y 292.81,Z 770.646,A -85,B 0,C 180,E1 22385.653,E2 22385.653} C_VEL
LIN {X 0,Y 296.208,Z 773.89,A -85,B 0,C 180,E1 22392.203,E2 22392.203} C_VEL
LIN {X 0,Y 297.034,Z 774.441,A -85,B 0,C 180,E1 22393.991,E2 22393.991} C_VEL
LIN {X 0,Y 296.422,Z 776.998,A -85,B 0,C 180,E1 22396.48,E2 22396.48} C_VEL
LIN {X 0,Y 294.243,Z 781.412,A -85,B 0,C 180,E1 22400.548,E2 22400.548} C_VEL
LIN {X 0,Y 294.288,Z 781.319,A -85,B 0,C 180,E1 22400.655,E2 22400.655} C_VEL
LIN {X 0,Y 295.814,Z 781.828,A -85,B 0,C 180,E1 22407.077,E2 22407.077} C_VEL
LIN {X 0,Y 295.814,Z 781.808,A -85,B 0,C 180,E1 22412.925,E2 22412.925} C_VEL
LIN {X 0,Y 294.403,Z 781.44,A -85,B 0,C 180,E1 22418.847,E2 22418.847} C_VEL
LIN {X 0,Y 292.038,Z 780.313,A -85,B 0,C 180,E1 22424.974,E2 22424.974} C_VEL
LIN {X 0,Y 288.703,Z 777.831,A -85,B 0,C 180,E1 22431.463,E2 22431.463} C_VEL
LIN {X 0,Y 284.638,Z 773.497,A -85,B 0,C 180,E1 22438.5,E2 22438.5} C_VEL
LIN {X 0,Y 278.528,Z 768.879,A -85,B 0,C 180,E1 22445.638,E2 22445.638} C_VEL
LIN {X 0,Y 273.347,Z 763.732,A -85,B 0,C 180,E1 22451.49,E2 22451.49} C_VEL
LIN {X 0,Y 266.093,Z 757.045,A -85,B 0,C 180,E1 22458.459,E2 22458.459} C_VEL
LIN {X 0,Y 257.835,Z 749.532,A -85,B 0,C 180,E1 22465.474,E2 22465.474} C_VEL
LIN {X 0,Y 245.773,Z 737.429,A -85,B 0,C 180,E1 22476.477,E2 22476.477} C_VEL
LIN {X 0,Y 241.819,Z 720.841,A -85,B 0,C 180,E1 22493.09,E2 22493.09} C_VEL
LIN {X 0,Y 242.627,Z 718.409,A -85,B 0,C 180,E1 22496.431,E2 22496.431} C_VEL
LIN {X 0,Y 243.267,Z 717.293,A -85,B 0,C 180,E1 22499.996,E2 22499.996} C_VEL
LIN {X 0,Y 242.824,Z 720.628,A -85,B 0,C 180,E1 22506.101,E2 22506.101} C_VEL
LIN {X 0,Y 242.478,Z 726.915,A -85,B 0,C 180,E1 22511.773,E2 22511.773} C_VEL
LIN {X 0,Y 241.331,Z 738.071,A -85,B 0,C 180,E1 22518.214,E2 22518.214} C_VEL
LIN {X 0,Y 235.233,Z 747.124,A -85,B 0,C 180,E1 22519.571,E2 22519.571} C_VEL
LIN {X 0,Y 209.915,Z 777.743,A -85,B 0,C 180,E1 22524.828,E2 22524.828} C_VEL
LIN {X 0,Y 184.641,Z 802.752,A -85,B 0,C 180,E1 22532.18,E2 22532.18} C_VEL
LIN {X 0,Y 162.544,Z 821.95,A -85,B 0,C 180,E1 22542.035,E2 22542.035} C_VEL
LIN {X 0,Y 145.489,Z 835.932,A -85,B 0,C 180,E1 22554.974,E2 22554.974} C_VEL
LIN {X 0,Y 136.037,Z 844.781,A -85,B 0,C 180,E1 22570.559,E2 22570.559} C_VEL
LIN {X 0,Y 133.814,Z 848.051,A -85,B 0,C 180,E1 22583.522,E2 22583.522} C_VEL
LIN {X 0,Y 133.991,Z 848.477,A -85,B 0,C 180,E1 22589.997,E2 22589.997} C_VEL
LIN {X 0,Y 134.485,Z 846.819,A -85,B 0,C 180,E1 22602.965,E2 22602.965} C_VEL
LIN {X 0,Y 140.653,Z 840.182,A -85,B 0,C 180,E1 22618.864,E2 22618.864} C_VEL
LIN {X 0,Y 155.773,Z 827.528,A -85,B 0,C 180,E1 22633.759,E2 22633.759} C_VEL
LIN {X 0,Y 177.218,Z 809.362,A -85,B 0,C 180,E1 22645.038,E2 22645.038} C_VEL
LIN {X 0,Y 201.222,Z 786.864,A -85,B 0,C 180,E1 22652.936,E2 22652.936} C_VEL
LIN {X 0,Y 226.59,Z 758.342,A -85,B 0,C 180,E1 22658.799,E2 22658.799} C_VEL
LIN {X 0,Y 240.43,Z 739.944,A -85,B 0,C 180,E1 22661.308,E2 22661.308} C_VEL
LIN {X 0,Y 241.512,Z 736.247,A -85,B 0,C 180,E1 22662.739,E2 22662.739} C_VEL
LIN {X 0,Y 242.461,Z 726.94,A -85,B 0,C 180,E1 22668.226,E2 22668.226} C_VEL
LIN {X 0,Y 242.713,Z 720.62,A -85,B 0,C 180,E1 22674.117,E2 22674.117} C_VEL
LIN {X 0,Y 243.264,Z 717.297,A -85,B 0,C 180,E1 22680.004,E2 22680.004} C_VEL
LIN {X 0,Y 242.288,Z 719.237,A -85,B 0,C 180,E1 22684.81,E2 22684.81} C_VEL
LIN {X 0,Y 241.4,Z 728.354,A -85,B 0,C 180,E1 22694.484,E2 22694.484} C_VEL
LIN {X 0,Y 255.114,Z 746.657,A -85,B 0,C 180,E1 22712.168,E2 22712.168} C_VEL
LIN {X 0,Y 264.684,Z 755.76,A -85,B 0,C 180,E1 22720.294,E2 22720.294} C_VEL
LIN {X 0,Y 271.113,Z 761.835,A -85,B 0,C 180,E1 22726.355,E2 22726.355} C_VEL
LIN {X 0,Y 276.883,Z 766.944,A -85,B 0,C 180,E1 22732.249,E2 22732.249} C_VEL
LIN {X 0,Y 282.422,Z 771.873,A -85,B 0,C 180,E1 22738.753,E2 22738.753} C_VEL
LIN {X 0,Y 286.91,Z 775.892,A -85,B 0,C 180,E1 22745.119,E2 22745.119} C_VEL
LIN {X 0,Y 290.404,Z 779.315,A -85,B 0,C 180,E1 22751.835,E2 22751.835} C_VEL
LIN {X 0,Y 293.402,Z 781.004,A -85,B 0,C 180,E1 22758.129,E2 22758.129} C_VEL
LIN {X 0,Y 294.288,Z 781.319,A -85,B 0,C 180,E1 22760.655,E2 22760.655} C_VEL
LIN {X 0,Y 293.411,Z 783.326,A -85,B 0,C 180,E1 22763.17,E2 22763.17} C_VEL
LIN {X 0,Y 290.012,Z 787.22,A -85,B 0,C 180,E1 22767.394,E2 22767.394} C_VEL
LIN {X 0,Y 290.026,Z 787.202,A -85,B 0,C 180,E1 22772.984,E2 22772.984} C_VEL
LIN {X 0,Y 288.564,Z 786.815,A -85,B 0,C 180,E1 22779.027,E2 22779.027} C_VEL
LIN {X 0,Y 286.004,Z 785.533,A -85,B 0,C 180,E1 22785.298,E2 22785.298} C_VEL
LIN {X 0,Y 282.586,Z 782.907,A -85,B 0,C 180,E1 22791.952,E2 22791.952} C_VEL
LIN {X 0,Y 279.919,Z 779.905,A -85,B 0,C 180,E1 22796.927,E2 22796.927} C_VEL
LIN {X 0,Y 273.841,Z 775.216,A -85,B 0,C 180,E1 22804.246,E2 22804.246} C_VEL
LIN {X 0,Y 268.637,Z 770.081,A -85,B 0,C 180,E1 22810.341,E2 22810.341} C_VEL
LIN {X 0,Y 260.453,Z 762.573,A -85,B 0,C 180,E1 22818.217,E2 22818.217} C_VEL
LIN {X 0,Y 251.585,Z 754.423,A -85,B 0,C 180,E1 22825.817,E2 22825.817} C_VEL
LIN {X 0,Y 237.65,Z 739.366,A -85,B 0,C 180,E1 22840.61,E2 22840.61} C_VEL
LIN {X 0,Y 237.022,Z 727.27,A -85,B 0,C 180,E1 22853.132,E2 22853.132} C_VEL
LIN {X 0,Y 237.851,Z 724.921,A -85,B 0,C 180,E1 22856.359,E2 22856.359} C_VEL
LIN {X 0,Y 238.606,Z 723.721,A -85,B 0,C 180,E1 22859.996,E2 22859.996} C_VEL
LIN {X 0,Y 238.068,Z 727.046,A -85,B 0,C 180,E1 22866.09,E2 22866.09} C_VEL
LIN {X 0,Y 237.387,Z 733.548,A -85,B 0,C 180,E1 22871.919,E2 22871.919} C_VEL
LIN {X 0,Y 236.145,Z 742.002,A -85,B 0,C 180,E1 22876.972,E2 22876.972} C_VEL
LIN {X 0,Y 211.232,Z 772.452,A -85,B 0,C 180,E1 22881.762,E2 22881.762} C_VEL
LIN {X 0,Y 185.316,Z 798.203,A -85,B 0,C 180,E1 22888.418,E2 22888.418} C_VEL
LIN {X 0,Y 160.107,Z 819.403,A -85,B 0,C 180,E1 22898.292,E2 22898.292} C_VEL
LIN {X 0,Y 140.198,Z 834.66,A -85,B 0,C 180,E1 22911.761,E2 22911.761} C_VEL
LIN {X 0,Y 128.47,Z 844.533,A -85,B 0,C 180,E1 22929.364,E2 22929.364} C_VEL
LIN {X 0,Y 125.909,Z 847.804,A -85,B 0,C 180,E1 22943.113,E2 22943.113} C_VEL
LIN {X 0,Y 126.076,Z 848.231,A -85,B 0,C 180,E1 22949.997,E2 22949.997} C_VEL
LIN {X 0,Y 126.688,Z 846.572,A -85,B 0,C 180,E1 22963.778,E2 22963.778} C_VEL
LIN {X 0,Y 133.6,Z 839.933,A -85,B 0,C 180,E1 22980.546,E2 22980.546} C_VEL
LIN {X 0,Y 150.852,Z 826.617,A -85,B 0,C 180,E1 22996.484,E2 22996.484} C_VEL
LIN {X 0,Y 175.284,Z 806.969,A -85,B 0,C 180,E1 23008.221,E2 23008.221} C_VEL
LIN {X 0,Y 200.121,Z 784.061,A -85,B 0,C 180,E1 23015.683,E2 23015.683} C_VEL
LIN {X 0,Y 225.402,Z 756.188,A -85,B 0,C 180,E1 23021.013,E2 23021.013} C_VEL
LIN {X 0,Y 236.062,Z 742.064,A -85,B 0,C 180,E1 23023.05,E2 23023.05} C_VEL
LIN {X 0,Y 237.517,Z 732.323,A -85,B 0,C 180,E1 23029.016,E2 23029.016} C_VEL
LIN {X 0,Y 238.21,Z 725.373,A -85,B 0,C 180,E1 23036.372,E2 23036.372} C_VEL
LIN {X 0,Y 238.605,Z 723.723,A -85,B 0,C 180,E1 23040.004,E2 23040.004} C_VEL
LIN {X 0,Y 237.492,Z 725.769,A -85,B 0,C 180,E1 23044.907,E2 23044.907} C_VEL
LIN {X 0,Y 236.898,Z 737.149,A -85,B 0,C 180,E1 23057.167,E2 23057.167} C_VEL
LIN {X 0,Y 250.117,Z 752.855,A -85,B 0,C 180,E1 23072.891,E2 23072.891} C_VEL
LIN {X 0,Y 259.482,Z 761.704,A -85,B 0,C 180,E1 23080.889,E2 23080.889} C_VEL
LIN {X 0,Y 266.364,Z 768.104,A -85,B 0,C 180,E1 23087.436,E2 23087.436} C_VEL
LIN {X 0,Y 271.686,Z 772.96,A -85,B 0,C 180,E1 23093,E2 23093} C_VEL
LIN {X 0,Y 278.195,Z 778.434,A -85,B 0,C 180,E1 23100.78,E2 23100.78} C_VEL
LIN {X 0,Y 281.373,Z 781.622,A -85,B 0,C 180,E1 23105.749,E2 23105.749} C_VEL
LIN {X 0,Y 284.906,Z 784.89,A -85,B 0,C 180,E1 23112.442,E2 23112.442} C_VEL
LIN {X 0,Y 287.464,Z 786.323,A -85,B 0,C 180,E1 23117.881,E2 23117.881} C_VEL
LIN {X 0,Y 289.538,Z 787.08,A -85,B 0,C 180,E1 23124.018,E2 23124.018} C_VEL
LIN {X 0,Y 290.012,Z 787.22,A -85,B 0,C 180,E1 23127.394,E2 23127.394} C_VEL
LIN {X 0,Y 287.03,Z 790,A -85,B 0,C 180,E1 23130.772,E2 23130.772} C_VEL
LIN {X 0,Y 283.681,Z 792.255,A -85,B 0,C 180,E1 23134.219,E2 23134.219} C_VEL
LIN {X 0,Y 282.471,Z 791.907,A -85,B 0,C 180,E1 23139.224,E2 23139.224} C_VEL
LIN {X 0,Y 279.791,Z 790.56,A -85,B 0,C 180,E1 23145.646,E2 23145.646} C_VEL
LIN {X 0,Y 276.284,Z 787.751,A -85,B 0,C 180,E1 23152.479,E2 23152.479} C_VEL
LIN {X 0,Y 273.136,Z 784.421,A -85,B 0,C 180,E1 23157.871,E2 23157.871} C_VEL
LIN {X 0,Y 266.959,Z 779.545,A -85,B 0,C 180,E1 23165.234,E2 23165.234} C_VEL
LIN {X 0,Y 261.505,Z 774.248,A -85,B 0,C 180,E1 23171.391,E2 23171.391} C_VEL
LIN {X 0,Y 253.47,Z 766.721,A -85,B 0,C 180,E1 23179.086,E2 23179.086} C_VEL
LIN {X 0,Y 243.69,Z 757.665,A -85,B 0,C 180,E1 23187.36,E2 23187.36} C_VEL
LIN {X 0,Y 231.868,Z 734.023,A -85,B 0,C 180,E1 23212.517,E2 23212.517} C_VEL
LIN {X 0,Y 232.932,Z 731.345,A -85,B 0,C 180,E1 23216.282,E2 23216.282} C_VEL
LIN {X 0,Y 233.857,Z 730.067,A -85,B 0,C 180,E1 23219.996,E2 23219.996} C_VEL
LIN {X 0,Y 233.19,Z 732.949,A -85,B 0,C 180,E1 23225.566,E2 23225.566} C_VEL
LIN {X 0,Y 232.251,Z 738.905,A -85,B 0,C 180,E1 23231.236,E2 23231.236} C_VEL
LIN {X 0,Y 230.438,Z 746.488,A -85,B 0,C 180,E1 23235.764,E2 23235.764} C_VEL
LIN {X 0,Y 203.637,Z 777.234,A -85,B 0,C 180,E1 23240.677,E2 23240.677} C_VEL
LIN {X 0,Y 175.59,Z 803.021,A -85,B 0,C 180,E1 23247.973,E2 23247.973} C_VEL
LIN {X 0,Y 152.085,Z 821.446,A -85,B 0,C 180,E1 23257.456,E2 23257.456} C_VEL
LIN {X 0,Y 130.722,Z 836.756,A -85,B 0,C 180,E1 23272.692,E2 23272.692} C_VEL
LIN {X 0,Y 120.931,Z 844.284,A -85,B 0,C 180,E1 23288.012,E2 23288.012} C_VEL
LIN {X 0,Y 118.007,Z 847.558,A -85,B 0,C 180,E1 23302.65,E2 23302.65} C_VEL
LIN {X 0,Y 118.174,Z 847.986,A -85,B 0,C 180,E1 23309.997,E2 23309.997} C_VEL
LIN {X 0,Y 118.907,Z 846.324,A -85,B 0,C 180,E1 23324.7,E2 23324.7} C_VEL
LIN {X 0,Y 126.288,Z 839.985,A -85,B 0,C 180,E1 23341.887,E2 23341.887} C_VEL
LIN {X 0,Y 143.234,Z 827.814,A -85,B 0,C 180,E1 23357.512,E2 23357.512} C_VEL
LIN {X 0,Y 167.033,Z 809.93,A -85,B 0,C 180,E1 23369.116,E2 23369.116} C_VEL
LIN {X 0,Y 194.346,Z 786.349,A -85,B 0,C 180,E1 23377.233,E2 23377.233} C_VEL
LIN {X 0,Y 221.265,Z 757.848,A -85,B 0,C 180,E1 23382.699,E2 23382.699} C_VEL
LIN {X 0,Y 230.863,Z 745.877,A -85,B 0,C 180,E1 23384.363,E2 23384.363} C_VEL
LIN {X 0,Y 232.567,Z 736.718,A -85,B 0,C 180,E1 23390.549,E2 23390.549} C_VEL
LIN {X 0,Y 233.324,Z 731.794,A -85,B 0,C 180,E1 23396.296,E2 23396.296} C_VEL
LIN {X 0,Y 233.84,Z 730.088,A -85,B 0,C 180,E1 23400.004,E2 23400.004} C_VEL
LIN {X 0,Y 232.352,Z 732.589,A -85,B 0,C 180,E1 23405.594,E2 23405.594} C_VEL
LIN {X 0,Y 242.321,Z 756.284,A -85,B 0,C 180,E1 23431.407,E2 23431.407} C_VEL
LIN {X 0,Y 252.105,Z 765.535,A -85,B 0,C 180,E1 23439.703,E2 23439.703} C_VEL
LIN {X 0,Y 259.3,Z 772.294,A -85,B 0,C 180,E1 23446.468,E2 23446.468} C_VEL
LIN {X 0,Y 265.409,Z 777.788,A -85,B 0,C 180,E1 23452.753,E2 23452.753} C_VEL
LIN {X 0,Y 271.497,Z 783.073,A -85,B 0,C 180,E1 23459.986,E2 23459.986} C_VEL
LIN {X 0,Y 275.029,Z 786.32,A -85,B 0,C 180,E1 23465.152,E2 23465.152} C_VEL
LIN {X 0,Y 278.065,Z 789.397,A -85,B 0,C 180,E1 23470.999,E2 23470.999} C_VEL
LIN {X 0,Y 281.364,Z 791.443,A -85,B 0,C 180,E1 23477.614,E2 23477.614} C_VEL
LIN {X 0,Y 283.454,Z 792.172,A -85,B 0,C 180,E1 23483.889,E2 23483.889} C_VEL
LIN {X 0,Y 284.241,Z 792.325,A -85,B 0,C 180,E1 23490.001,E2 23490.001} C_VEL
LIN {X 0,Y 283.681,Z 792.255,A -85,B 0,C 180,E1 23494.219,E2 23494.219} C_VEL
LIN {X 0,Y 281.104,Z 793.971,A -85,B 0,C 180,E1 23496.804,E2 23496.804} C_VEL
LIN {X 0,Y 275.478,Z 796.636,A -85,B 0,C 180,E1 23501.041,E2 23501.041} C_VEL
LIN {X 0,Y 275.427,Z 796.495,A -85,B 0,C 180,E1 23501.155,E2 23501.155} C_VEL
LIN {X 0,Y 273.398,Z 795.378,A -85,B 0,C 180,E1 23506.022,E2 23506.022} C_VEL
LIN {X 0,Y 269.738,Z 792.242,A -85,B 0,C 180,E1 23513.056,E2 23513.056} C_VEL
LIN {X 0,Y 266.26,Z 788.791,A -85,B 0,C 180,E1 23518.656,E2 23518.656} C_VEL
LIN {X 0,Y 260.297,Z 783.982,A -85,B 0,C 180,E1 23525.741,E2 23525.741} C_VEL
LIN {X 0,Y 254.317,Z 778.286,A -85,B 0,C 180,E1 23532.294,E2 23532.294} C_VEL
LIN {X 0,Y 245.619,Z 770.096,A -85,B 0,C 180,E1 23540.513,E2 23540.513} C_VEL
LIN {X 0,Y 235.538,Z 760.833,A -85,B 0,C 180,E1 23549.163,E2 23549.163} C_VEL
LIN {X 0,Y 227.342,Z 738.629,A -85,B 0,C 180,E1 23574.669,E2 23574.669} C_VEL
LIN {X 0,Y 228.853,Z 736.227,A -85,B 0,C 180,E1 23579.996,E2 23579.996} C_VEL
LIN {X 0,Y 227.916,Z 740.094,A -85,B 0,C 180,E1 23586.702,E2 23586.702} C_VEL
LIN {X 0,Y 226.252,Z 747.497,A -85,B 0,C 180,E1 23592.927,E2 23592.927} C_VEL
LIN {X 0,Y 225.064,Z 750.327,A -85,B 0,C 180,E1 23594.313,E2 23594.313} C_VEL
LIN {X 0,Y 199.299,Z 778.523,A -85,B 0,C 180,E1 23598.829,E2 23598.829} C_VEL
LIN {X 0,Y 170.007,Z 804.333,A -85,B 0,C 180,E1 23606.153,E2 23606.153} C_VEL
LIN {X 0,Y 144.814,Z 822.832,A -85,B 0,C 180,E1 23616.136,E2 23616.136} C_VEL
LIN {X 0,Y 124.328,Z 836.501,A -85,B 0,C 180,E1 23630.412,E2 23630.412} C_VEL
LIN {X 0,Y 113.486,Z 844.035,A -85,B 0,C 180,E1 23646.486,E2 23646.486} C_VEL
LIN {X 0,Y 110.109,Z 847.311,A -85,B 0,C 180,E1 23662.119,E2 23662.119} C_VEL
LIN {X 0,Y 110.255,Z 847.74,A -85,B 0,C 180,E1 23669.996,E2 23669.996} C_VEL
LIN {X 0,Y 111.168,Z 846.076,A -85,B 0,C 180,E1 23685.749,E2 23685.749} C_VEL
LIN {X 0,Y 119.256,Z 839.88,A -85,B 0,C 180,E1 23703.683,E2 23703.683} C_VEL
LIN {X 0,Y 137.833,Z 827.562,A -85,B 0,C 180,E1 23720.024,E2 23720.024} C_VEL
LIN {X 0,Y 163.014,Z 809.681,A -85,B 0,C 180,E1 23731.566,E2 23731.566} C_VEL
LIN {X 0,Y 190.804,Z 786.607,A -85,B 0,C 180,E1 23739.356,E2 23739.356} C_VEL
LIN {X 0,Y 219.001,Z 757.602,A -85,B 0,C 180,E1 23744.715,E2 23744.715} C_VEL
LIN {X 0,Y 225.023,Z 750.398,A -85,B 0,C 180,E1 23745.663,E2 23745.663} C_VEL
LIN {X 0,Y 226.749,Z 745.5,A -85,B 0,C 180,E1 23748.488,E2 23748.488} C_VEL
LIN {X 0,Y 228.04,Z 738.966,A -85,B 0,C 180,E1 23754.866,E2 23754.866} C_VEL
LIN {X 0,Y 228.819,Z 736.268,A -85,B 0,C 180,E1 23760.004,E2 23760.004} C_VEL
LIN {X 0,Y 227.347,Z 738.64,A -85,B 0,C 180,E1 23765.383,E2 23765.383} C_VEL
LIN {X 0,Y 235.605,Z 760.758,A -85,B 0,C 180,E1 23790.827,E2 23790.827} C_VEL
LIN {X 0,Y 245.562,Z 770.106,A -85,B 0,C 180,E1 23799.467,E2 23799.467} C_VEL
LIN {X 0,Y 254.35,Z 778.312,A -85,B 0,C 180,E1 23807.729,E2 23807.729} C_VEL
LIN {X 0,Y 260.753,Z 784.22,A -85,B 0,C 180,E1 23814.642,E2 23814.642} C_VEL
LIN {X 0,Y 266.287,Z 788.801,A -85,B 0,C 180,E1 23821.354,E2 23821.354} C_VEL
LIN {X 0,Y 269.769,Z 792.291,A -85,B 0,C 180,E1 23826.95,E2 23826.95} C_VEL
LIN {X 0,Y 273.393,Z 795.39,A -85,B 0,C 180,E1 23833.981,E2 23833.981} C_VEL
LIN {X 0,Y 276.278,Z 796.735,A -85,B 0,C 180,E1 23840.571,E2 23840.571} C_VEL
LIN {X 0,Y 277.817,Z 797.279,A -85,B 0,C 180,E1 23846.888,E2 23846.888} C_VEL
LIN {X 0,Y 277.814,Z 797.261,A -85,B 0,C 180,E1 23853.115,E2 23853.115} C_VEL
LIN {X 0,Y 275.909,Z 796.702,A -85,B 0,C 180,E1 23860.1,E2 23860.1} C_VEL
LIN {X 0,Y 275.427,Z 796.495,A -85,B 0,C 180,E1 23861.155,E2 23861.155} C_VEL
LIN {X 0,Y 272.226,Z 797.697,A -85,B 0,C 180,E1 23863.809,E2 23863.809} C_VEL
LIN {X 0,Y 265.73,Z 799.303,A -85,B 0,C 180,E1 23868.17,E2 23868.17} C_VEL
LIN {X 0,Y 265.666,Z 799.141,A -85,B 0,C 180,E1 23868.288,E2 23868.288} C_VEL
LIN {X 0,Y 261.713,Z 795.016,A -85,B 0,C 180,E1 23876.079,E2 23876.079} C_VEL
LIN {X 0,Y 257.227,Z 791.439,A -85,B 0,C 180,E1 23881.871,E2 23881.871} C_VEL
LIN {X 0,Y 251.342,Z 786.007,A -85,B 0,C 180,E1 23888.689,E2 23888.689} C_VEL
LIN {X 0,Y 244.793,Z 780.153,A -85,B 0,C 180,E1 23895.241,E2 23895.241} C_VEL
LIN {X 0,Y 238.842,Z 774.415,A -85,B 0,C 180,E1 23900.813,E2 23900.813} C_VEL
LIN {X 0,Y 227.866,Z 764.545,A -85,B 0,C 180,E1 23910.587,E2 23910.587} C_VEL
LIN {X 0,Y 221.996,Z 744.78,A -85,B 0,C 180,E1 23934.541,E2 23934.541} C_VEL
LIN {X 0,Y 223.731,Z 742.333,A -85,B 0,C 180,E1 23939.996,E2 23939.996} C_VEL
LIN {X 0,Y 222.775,Z 745.429,A -85,B 0,C 180,E1 23945.829,E2 23945.829} C_VEL
LIN {X 0,Y 220.794,Z 752.673,A -85,B 0,C 180,E1 23952.327,E2 23952.327} C_VEL
LIN {X 0,Y 217.002,Z 757.338,A -85,B 0,C 180,E1 23953.2,E2 23953.2} C_VEL
LIN {X 0,Y 188.591,Z 785.901,A -85,B 0,C 180,E1 23958.219,E2 23958.219} C_VEL
LIN {X 0,Y 158.912,Z 809.731,A -85,B 0,C 180,E1 23966.005,E2 23966.005} C_VEL
LIN {X 0,Y 132.773,Z 827.307,A -85,B 0,C 180,E1 23977.286,E2 23977.286} C_VEL
LIN {X 0,Y 113.344,Z 839.103,A -85,B 0,C 180,E1 23993.002,E2 23993.002} C_VEL
LIN {X 0,Y 103.485,Z 845.828,A -85,B 0,C 180,E1 24013.04,E2 24013.04} C_VEL
LIN {X 0,Y 102.343,Z 847.494,A -85,B 0,C 180,E1 24029.996,E2 24029.996} C_VEL
LIN {X 0,Y 103.489,Z 845.829,A -85,B 0,C 180,E1 24046.951,E2 24046.951} C_VEL
LIN {X 0,Y 113.468,Z 839.052,A -85,B 0,C 180,E1 24067.081,E2 24067.081} C_VEL
LIN {X 0,Y 135.144,Z 825.857,A -85,B 0,C 180,E1 24084.045,E2 24084.045} C_VEL
LIN {X 0,Y 164.299,Z 805.791,A -85,B 0,C 180,E1 24095.71,E2 24095.71} C_VEL
LIN {X 0,Y 193.517,Z 781.32,A -85,B 0,C 180,E1 24102.784,E2 24102.784} C_VEL
LIN {X 0,Y 220.108,Z 753.823,A -85,B 0,C 180,E1 24107.233,E2 24107.233} C_VEL
LIN {X 0,Y 221.996,Z 748.229,A -85,B 0,C 180,E1 24111.207,E2 24111.207} C_VEL
LIN {X 0,Y 223.033,Z 744.175,A -85,B 0,C 180,E1 24116.125,E2 24116.125} C_VEL
LIN {X 0,Y 223.711,Z 742.356,A -85,B 0,C 180,E1 24120.004,E2 24120.004} C_VEL
LIN {X 0,Y 222.004,Z 744.787,A -85,B 0,C 180,E1 24125.513,E2 24125.513} C_VEL
LIN {X 0,Y 230.229,Z 766.431,A -85,B 0,C 180,E1 24151.629,E2 24151.629} C_VEL
LIN {X 0,Y 239.991,Z 775.512,A -85,B 0,C 180,E1 24160.226,E2 24160.226} C_VEL
LIN {X 0,Y 248.23,Z 783.162,A -85,B 0,C 180,E1 24168.036,E2 24168.036} C_VEL
LIN {X 0,Y 253.305,Z 787.86,A -85,B 0,C 180,E1 24173.437,E2 24173.437} C_VEL
LIN {X 0,Y 259.396,Z 793.067,A -85,B 0,C 180,E1 24180.769,E2 24180.769} C_VEL
LIN {X 0,Y 263.13,Z 796.67,A -85,B 0,C 180,E1 24186.58,E2 24186.58} C_VEL
LIN {X 0,Y 266.938,Z 799.98,A -85,B 0,C 180,E1 24193.958,E2 24193.958} C_VEL
LIN {X 0,Y 269.802,Z 801.419,A -85,B 0,C 180,E1 24200.342,E2 24200.342} C_VEL
LIN {X 0,Y 271.444,Z 801.948,A -85,B 0,C 180,E1 24206.815,E2 24206.815} C_VEL
LIN {X 0,Y 271.443,Z 801.927,A -85,B 0,C 180,E1 24213.188,E2 24213.188} C_VEL
LIN {X 0,Y 269.711,Z 801.413,A -85,B 0,C 180,E1 24219.664,E2 24219.664} C_VEL
LIN {X 0,Y 266.731,Z 799.839,A -85,B 0,C 180,E1 24226.433,E2 24226.433} C_VEL
LIN {X 0,Y 265.666,Z 799.141,A -85,B 0,C 180,E1 24228.288,E2 24228.288} C_VEL
LIN {X 0,Y 260.531,Z 799.718,A -85,B 0,C 180,E1 24231.929,E2 24231.929} C_VEL
LIN {X 0,Y 255.128,Z 799.63,A -85,B 0,C 180,E1 24235.672,E2 24235.672} C_VEL
LIN {X 0,Y 250.142,Z 795.454,A -85,B 0,C 180,E1 24242.369,E2 24242.369} C_VEL
LIN {X 0,Y 242.96,Z 788.775,A -85,B 0,C 180,E1 24250.6,E2 24250.6} C_VEL
LIN {X 0,Y 234.698,Z 781.083,A -85,B 0,C 180,E1 24258.609,E2 24258.609} C_VEL
LIN {X 0,Y 224.744,Z 772.026,A -85,B 0,C 180,E1 24267.506,E2 24267.506} C_VEL
LIN {X 0,Y 216.324,Z 751.099,A -85,B 0,C 180,E1 24293.99,E2 24293.99} C_VEL
LIN {X 0,Y 218.401,Z 748.273,A -85,B 0,C 180,E1 24299.996,E2 24299.996} C_VEL
LIN {X 0,Y 217.287,Z 751.481,A -85,B 0,C 180,E1 24305.975,E2 24305.975} C_VEL
LIN {X 0,Y 215.289,Z 757.089,A -85,B 0,C 180,E1 24311.09,E2 24311.09} C_VEL
LIN {X 0,Y 186.21,Z 785.649,A -85,B 0,C 180,E1 24315.84,E2 24315.84} C_VEL
LIN {X 0,Y 156.449,Z 808.8,A -85,B 0,C 180,E1 24322.996,E2 24322.996} C_VEL
LIN {X 0,Y 127.986,Z 827.056,A -85,B 0,C 180,E1 24334.372,E2 24334.372} C_VEL
LIN {X 0,Y 106.943,Z 838.852,A -85,B 0,C 180,E1 24350.372,E2 24350.372} C_VEL
LIN {X 0,Y 95.821,Z 845.58,A -85,B 0,C 180,E1 24371.637,E2 24371.637} C_VEL
LIN {X 0,Y 94.42,Z 847.248,A -85,B 0,C 180,E1 24389.996,E2 24389.996} C_VEL
LIN {X 0,Y 96.18,Z 845.326,A -85,B 0,C 180,E1 24409.749,E2 24409.749} C_VEL
LIN {X 0,Y 107.067,Z 838.801,A -85,B 0,C 180,E1 24429.716,E2 24429.716} C_VEL
LIN {X 0,Y 130.517,Z 825.604,A -85,B 0,C 180,E1 24446.948,E2 24446.948} C_VEL
LIN {X 0,Y 159.615,Z 806.58,A -85,B 0,C 180,E1 24457.935,E2 24457.935} C_VEL
LIN {X 0,Y 187.91,Z 784.096,A -85,B 0,C 180,E1 24464.498,E2 24464.498} C_VEL
LIN {X 0,Y 215.301,Z 757.107,A -85,B 0,C 180,E1 24468.874,E2 24468.874} C_VEL
LIN {X 0,Y 217.163,Z 751.619,A -85,B 0,C 180,E1 24474.021,E2 24474.021} C_VEL
LIN {X 0,Y 218.382,Z 748.294,A -85,B 0,C 180,E1 24480.004,E2 24480.004} C_VEL
LIN {X 0,Y 216.348,Z 751.073,A -85,B 0,C 180,E1 24486.01,E2 24486.01} C_VEL
LIN {X 0,Y 224.774,Z 771.999,A -85,B 0,C 180,E1 24512.489,E2 24512.489} C_VEL
LIN {X 0,Y 234.672,Z 781.106,A -85,B 0,C 180,E1 24521.393,E2 24521.393} C_VEL
LIN {X 0,Y 243.025,Z 788.742,A -85,B 0,C 180,E1 24529.419,E2 24529.419} C_VEL
LIN {X 0,Y 249.724,Z 795.04,A -85,B 0,C 180,E1 24537.056,E2 24537.056} C_VEL
LIN {X 0,Y 254.337,Z 798.77,A -85,B 0,C 180,E1 24542.875,E2 24542.875} C_VEL
LIN {X 0,Y 257.975,Z 802.595,A -85,B 0,C 180,E1 24549.455,E2 24549.455} C_VEL
LIN {X 0,Y 261.652,Z 805.173,A -85,B 0,C 180,E1 24556.664,E2 24556.664} C_VEL
LIN {X 0,Y 264.179,Z 806.147,A -85,B 0,C 180,E1 24563.442,E2 24563.442} C_VEL
LIN {X 0,Y 265.152,Z 806.349,A -85,B 0,C 180,E1 24570.002,E2 24570.002} C_VEL
LIN {X 0,Y 264.124,Z 806.14,A -85,B 0,C 180,E1 24576.563,E2 24576.563} C_VEL
LIN {X 0,Y 261.607,Z 805.135,A -85,B 0,C 180,E1 24583.342,E2 24583.342} C_VEL
LIN {X 0,Y 257.98,Z 802.551,A -85,B 0,C 180,E1 24590.62,E2 24590.62} C_VEL
LIN {X 0,Y 255.128,Z 799.63,A -85,B 0,C 180,E1 24595.672,E2 24595.672} C_VEL
LIN {X 0,Y 251.023,Z 799.417,A -85,B 0,C 180,E1 24598.491,E2 24598.491} C_VEL
LIN {X 0,Y 242.723,Z 799.163,A -85,B 0,C 180,E1 24603.001,E2 24603.001} C_VEL
LIN {X 0,Y 242.493,Z 798.901,A -85,B 0,C 180,E1 24603.256,E2 24603.256} C_VEL
LIN {X 0,Y 236.659,Z 793.304,A -85,B 0,C 180,E1 24610.074,E2 24610.074} C_VEL
LIN {X 0,Y 229.652,Z 786.92,A -85,B 0,C 180,E1 24616.962,E2 24616.962} C_VEL
LIN {X 0,Y 219.161,Z 777.371,A -85,B 0,C 180,E1 24626.572,E2 24626.572} C_VEL
LIN {X 0,Y 210.575,Z 757.046,A -85,B 0,C 180,E1 24653.722,E2 24653.722} C_VEL
LIN {X 0,Y 212.943,Z 754.09,A -85,B 0,C 180,E1 24659.996,E2 24659.996} C_VEL
LIN {X 0,Y 211.64,Z 757.241,A -85,B 0,C 180,E1 24665.93,E2 24665.93} C_VEL
LIN {X 0,Y 210.554,Z 760.003,A -85,B 0,C 180,E1 24668.875,E2 24668.875} C_VEL
LIN {X 0,Y 207.375,Z 763.712,A -85,B 0,C 180,E1 24669.821,E2 24669.821} C_VEL
LIN {X 0,Y 177.892,Z 790.514,A -85,B 0,C 180,E1 24674.571,E2 24674.571} C_VEL
LIN {X 0,Y 146.643,Z 813.064,A -85,B 0,C 180,E1 24682.153,E2 24682.153} C_VEL
LIN {X 0,Y 118.321,Z 829.612,A -85,B 0,C 180,E1 24694,E2 24694} C_VEL
LIN {X 0,Y 97.202,Z 840.436,A -85,B 0,C 180,E1 24711.607,E2 24711.607} C_VEL
LIN {X 0,Y 88.248,Z 845.332,A -85,B 0,C 180,E1 24729.997,E2 24729.997} C_VEL
LIN {X 0,Y 86.495,Z 847.002,A -85,B 0,C 180,E1 24749.995,E2 24749.995} C_VEL
LIN {X 0,Y 88.254,Z 845.334,A -85,B 0,C 180,E1 24769.992,E2 24769.992} C_VEL
LIN {X 0,Y 101.211,Z 838.409,A -85,B 0,C 180,E1 24792.959,E2 24792.959} C_VEL
LIN {X 0,Y 125.904,Z 825.545,A -85,B 0,C 180,E1 24809.882,E2 24809.882} C_VEL
LIN {X 0,Y 156.957,Z 806.176,A -85,B 0,C 180,E1 24820.764,E2 24820.764} C_VEL
LIN {X 0,Y 187.618,Z 782.333,A -85,B 0,C 180,E1 24827.207,E2 24827.207} C_VEL
LIN {X 0,Y 209.092,Z 761.933,A -85,B 0,C 180,E1 24830.379,E2 24830.379} C_VEL
LIN {X 0,Y 210.791,Z 759.352,A -85,B 0,C 180,E1 24831.773,E2 24831.773} C_VEL
LIN {X 0,Y 212.017,Z 756.074,A -85,B 0,C 180,E1 24835.923,E2 24835.923} C_VEL
LIN {X 0,Y 212.928,Z 754.106,A -85,B 0,C 180,E1 24840.004,E2 24840.004} C_VEL
LIN {X 0,Y 210.757,Z 756.765,A -85,B 0,C 180,E1 24845.905,E2 24845.905} C_VEL
LIN {X 0,Y 217.215,Z 775.608,A -85,B 0,C 180,E1 24871.406,E2 24871.406} C_VEL
LIN {X 0,Y 227.97,Z 785.271,A -85,B 0,C 180,E1 24881.452,E2 24881.452} C_VEL
LIN {X 0,Y 236.722,Z 793.28,A -85,B 0,C 180,E1 24889.908,E2 24889.908} C_VEL
LIN {X 0,Y 241.94,Z 798.251,A -85,B 0,C 180,E1 24895.853,E2 24895.853} C_VEL
LIN {X 0,Y 247.526,Z 802.852,A -85,B 0,C 180,E1 24902.808,E2 24902.808} C_VEL
LIN {X 0,Y 250.906,Z 806.365,A -85,B 0,C 180,E1 24908.849,E2 24908.849} C_VEL
LIN {X 0,Y 254.683,Z 809.179,A -85,B 0,C 180,E1 24916.292,E2 24916.292} C_VEL
LIN {X 0,Y 257.406,Z 810.307,A -85,B 0,C 180,E1 24923.268,E2 24923.268} C_VEL
LIN {X 0,Y 258.488,Z 810.559,A -85,B 0,C 180,E1 24930.002,E2 24930.002} C_VEL
LIN {X 0,Y 257.347,Z 810.297,A -85,B 0,C 180,E1 24936.736,E2 24936.736} C_VEL
LIN {X 0,Y 254.65,Z 809.152,A -85,B 0,C 180,E1 24943.713,E2 24943.713} C_VEL
LIN {X 0,Y 250.914,Z 806.357,A -85,B 0,C 180,E1 24951.154,E2 24951.154} C_VEL
LIN {X 0,Y 247.103,Z 802.462,A -85,B 0,C 180,E1 24957.754,E2 24957.754} C_VEL
LIN {X 0,Y 242.493,Z 798.901,A -85,B 0,C 180,E1 24963.256,E2 24963.256} C_VEL
LIN {X 0,Y 237.874,Z 797.952,A -85,B 0,C 180,E1 24966.18,E2 24966.18} C_VEL
LIN {X 0,Y 228.709,Z 796.243,A -85,B 0,C 180,E1 24971.125,E2 24971.125} C_VEL
LIN {X 0,Y 220.755,Z 788.894,A -85,B 0,C 180,E1 24978.76,E2 24978.76} C_VEL
LIN {X 0,Y 209.516,Z 779.298,A -85,B 0,C 180,E1 24989.805,E2 24989.805} C_VEL
LIN {X 0,Y 205.681,Z 761.378,A -85,B 0,C 180,E1 25015.788,E2 25015.788} C_VEL
LIN {X 0,Y 207.291,Z 759.74,A -85,B 0,C 180,E1 25019.996,E2 25019.996} C_VEL
LIN {X 0,Y 205.729,Z 763.139,A -85,B 0,C 180,E1 25026.243,E2 25026.243} C_VEL
LIN {X 0,Y 204.366,Z 765.267,A -85,B 0,C 180,E1 25027.827,E2 25027.827} C_VEL
LIN {X 0,Y 172.374,Z 793.12,A -85,B 0,C 180,E1 25032.645,E2 25032.645} C_VEL
LIN {X 0,Y 140.573,Z 814.696,A -85,B 0,C 180,E1 25040.059,E2 25040.059} C_VEL
LIN {X 0,Y 111.282,Z 830.734,A -85,B 0,C 180,E1 25052.051,E2 25052.051} C_VEL
LIN {X 0,Y 87.635,Z 841.677,A -85,B 0,C 180,E1 25072.932,E2 25072.932} C_VEL
LIN {X 0,Y 80.115,Z 845.359,A -85,B 0,C 180,E1 25090.317,E2 25090.317} C_VEL
LIN {X 0,Y 78.568,Z 846.755,A -85,B 0,C 180,E1 25109.995,E2 25109.995} C_VEL
LIN {X 0,Y 80.728,Z 845.085,A -85,B 0,C 180,E1 25131.948,E2 25131.948} C_VEL
LIN {X 0,Y 94.825,Z 838.432,A -85,B 0,C 180,E1 25155.728,E2 25155.728} C_VEL
LIN {X 0,Y 121.817,Z 825.386,A -85,B 0,C 180,E1 25173.122,E2 25173.122} C_VEL
LIN {X 0,Y 154.479,Z 805.911,A -85,B 0,C 180,E1 25183.632,E2 25183.632} C_VEL
LIN {X 0,Y 185.766,Z 782.272,A -85,B 0,C 180,E1 25189.617,E2 25189.617} C_VEL
LIN {X 0,Y 204.332,Z 765.311,A -85,B 0,C 180,E1 25192.152,E2 25192.152} C_VEL
LIN {X 0,Y 205.603,Z 763.258,A -85,B 0,C 180,E1 25193.758,E2 25193.758} C_VEL
LIN {X 0,Y 207.277,Z 759.754,A -85,B 0,C 180,E1 25200.004,E2 25200.004} C_VEL
LIN {X 0,Y 204.757,Z 762.695,A -85,B 0,C 180,E1 25206.351,E2 25206.351} C_VEL
LIN {X 0,Y 211.535,Z 780.851,A -85,B 0,C 180,E1 25232.347,E2 25232.347} C_VEL
LIN {X 0,Y 220.757,Z 788.899,A -85,B 0,C 180,E1 25241.246,E2 25241.246} C_VEL
LIN {X 0,Y 229.592,Z 796.971,A -85,B 0,C 180,E1 25249.69,E2 25249.69} C_VEL
LIN {X 0,Y 235.453,Z 802.51,A -85,B 0,C 180,E1 25256.431,E2 25256.431} C_VEL
LIN {X 0,Y 241.376,Z 807.52,A -85,B 0,C 180,E1 25264.05,E2 25264.05} C_VEL
LIN {X 0,Y 245.641,Z 811.693,A -85,B 0,C 180,E1 25272.114,E2 25272.114} C_VEL
LIN {X 0,Y 249.197,Z 813.774,A -85,B 0,C 180,E1 25279.535,E2 25279.535} C_VEL
LIN {X 0,Y 251.246,Z 814.442,A -85,B 0,C 180,E1 25286.558,E2 25286.558} C_VEL
LIN {X 0,Y 251.608,Z 814.44,A -85,B 0,C 180,E1 25290.002,E2 25290.002} C_VEL
LIN {X 0,Y 250.416,Z 814.228,A -85,B 0,C 180,E1 25296.924,E2 25296.924} C_VEL
LIN {X 0,Y 247.508,Z 812.907,A -85,B 0,C 180,E1 25304.117,E2 25304.117} C_VEL
LIN {X 0,Y 243.621,Z 809.874,A -85,B 0,C 180,E1 25311.819,E2 25311.819} C_VEL
LIN {X 0,Y 239.795,Z 806.074,A -85,B 0,C 180,E1 25318.23,E2 25318.23} C_VEL
LIN {X 0,Y 233.674,Z 801.049,A -85,B 0,C 180,E1 25325.537,E2 25325.537} C_VEL
LIN {X 0,Y 228.709,Z 796.243,A -85,B 0,C 180,E1 25331.125,E2 25331.125} C_VEL
LIN {X 0,Y 223.455,Z 794.656,A -85,B 0,C 180,E1 25334.139,E2 25334.139} C_VEL
LIN {X 0,Y 213.137,Z 792.111,A -85,B 0,C 180,E1 25339.26,E2 25339.26} C_VEL
LIN {X 0,Y 203.777,Z 784.357,A -85,B 0,C 180,E1 25348.773,E2 25348.773} C_VEL
LIN {X 0,Y 199.718,Z 766.952,A -85,B 0,C 180,E1 25375.662,E2 25375.662} C_VEL
LIN {X 0,Y 201.527,Z 765.289,A -85,B 0,C 180,E1 25379.995,E2 25379.995} C_VEL
LIN {X 0,Y 199.946,Z 768.204,A -85,B 0,C 180,E1 25385.723,E2 25385.723} C_VEL
LIN {X 0,Y 170.313,Z 793.231,A -85,B 0,C 180,E1 25390.064,E2 25390.064} C_VEL
LIN {X 0,Y 137.992,Z 814.444,A -85,B 0,C 180,E1 25396.881,E2 25396.881} C_VEL
LIN {X 0,Y 107.166,Z 830.478,A -85,B 0,C 180,E1 25408.341,E2 25408.341} C_VEL
LIN {X 0,Y 84.137,Z 840.278,A -85,B 0,C 180,E1 25425.824,E2 25425.824} C_VEL
LIN {X 0,Y 73.303,Z 844.835,A -85,B 0,C 180,E1 25445.681,E2 25445.681} C_VEL
LIN {X 0,Y 70.667,Z 846.51,A -85,B 0,C 180,E1 25469.994,E2 25469.994} C_VEL
LIN {X 0,Y 73.314,Z 844.836,A -85,B 0,C 180,E1 25494.303,E2 25494.303} C_VEL
LIN {X 0,Y 89.332,Z 838.182,A -85,B 0,C 180,E1 25519.47,E2 25519.47} C_VEL
LIN {X 0,Y 115.906,Z 826.304,A -85,B 0,C 180,E1 25535.684,E2 25535.684} C_VEL
LIN {X 0,Y 147.019,Z 809.041,A -85,B 0,C 180,E1 25545.387,E2 25545.387} C_VEL
LIN {X 0,Y 178.977,Z 786.546,A -85,B 0,C 180,E1 25551.313,E2 25551.313} C_VEL
LIN {X 0,Y 199.831,Z 768.303,A -85,B 0,C 180,E1 25554.282,E2 25554.282} C_VEL
LIN {X 0,Y 201.517,Z 765.299,A -85,B 0,C 180,E1 25560.005,E2 25560.005} C_VEL
LIN {X 0,Y 198.106,Z 769.203,A -85,B 0,C 180,E1 25568.028,E2 25568.028} C_VEL
LIN {X 0,Y 205.756,Z 785.903,A -85,B 0,C 180,E1 25593.375,E2 25593.375} C_VEL
LIN {X 0,Y 215.101,Z 793.932,A -85,B 0,C 180,E1 25602.581,E2 25602.581} C_VEL
LIN {X 0,Y 223.084,Z 801.115,A -85,B 0,C 180,E1 25610.321,E2 25610.321} C_VEL
LIN {X 0,Y 230.109,Z 807.546,A -85,B 0,C 180,E1 25618.492,E2 25618.492} C_VEL
LIN {X 0,Y 234.467,Z 811.236,A -85,B 0,C 180,E1 25624.3,E2 25624.3} C_VEL
LIN {X 0,Y 238.342,Z 815.114,A -85,B 0,C 180,E1 25631.758,E2 25631.758} C_VEL
LIN {X 0,Y 242.002,Z 817.341,A -85,B 0,C 180,E1 25639.22,E2 25639.22} C_VEL
LIN {X 0,Y 244.197,Z 818.044,A -85,B 0,C 180,E1 25646.459,E2 25646.459} C_VEL
LIN {X 0,Y 244.606,Z 818.056,A -85,B 0,C 180,E1 25650.002,E2 25650.002} C_VEL
LIN {X 0,Y 243.249,Z 817.793,A -85,B 0,C 180,E1 25657.129,E2 25657.129} C_VEL
LIN {X 0,Y 240.208,Z 816.438,A -85,B 0,C 180,E1 25664.555,E2 25664.555} C_VEL
LIN {X 0,Y 236.175,Z 813.11,A -85,B 0,C 180,E1 25672.544,E2 25672.544} C_VEL
LIN {X 0,Y 231.859,Z 809.045,A -85,B 0,C 180,E1 25679.288,E2 25679.288} C_VEL
LIN {X 0,Y 225.326,Z 803.399,A -85,B 0,C 180,E1 25687.068,E2 25687.068} C_VEL
LIN {X 0,Y 218.396,Z 796.984,A -85,B 0,C 180,E1 25694.257,E2 25694.257} C_VEL
LIN {X 0,Y 213.137,Z 792.111,A -85,B 0,C 180,E1 25699.26,E2 25699.26} C_VEL
LIN {X 0,Y 207.503,Z 790.484,A -85,B 0,C 180,E1 25702.457,E2 25702.457} C_VEL
LIN {X 0,Y 197.62,Z 789.054,A -85,B 0,C 180,E1 25708.047,E2 25708.047} C_VEL
LIN {X 0,Y 193.58,Z 772.376,A -85,B 0,C 180,E1 25735.524,E2 25735.524} C_VEL
LIN {X 0,Y 195.536,Z 770.61,A -85,B 0,C 180,E1 25739.995,E2 25739.995} C_VEL
LIN {X 0,Y 194.583,Z 772.249,A -85,B 0,C 180,E1 25743.886,E2 25743.886} C_VEL
LIN {X 0,Y 163.654,Z 796.841,A -85,B 0,C 180,E1 25748.174,E2 25748.174} C_VEL
LIN {X 0,Y 129.074,Z 817.95,A -85,B 0,C 180,E1 25755.298,E2 25755.298} C_VEL
LIN {X 0,Y 96.414,Z 833.167,A -85,B 0,C 180,E1 25767.993,E2 25767.993} C_VEL
LIN {X 0,Y 71.62,Z 842.54,A -85,B 0,C 180,E1 25790.789,E2 25790.789} C_VEL
LIN {X 0,Y 63.054,Z 845.828,A -85,B 0,C 180,E1 25816.147,E2 25816.147} C_VEL
LIN {X 0,Y 62.734,Z 846.264,A -85,B 0,C 180,E1 25829.994,E2 25829.994} C_VEL
LIN {X 0,Y 66.071,Z 844.588,A -85,B 0,C 180,E1 25857.173,E2 25857.173} C_VEL
LIN {X 0,Y 84.254,Z 837.931,A -85,B 0,C 180,E1 25883.695,E2 25883.695} C_VEL
LIN {X 0,Y 112.79,Z 826.049,A -85,B 0,C 180,E1 25899.466,E2 25899.466} C_VEL
LIN {X 0,Y 146.037,Z 808.262,A -85,B 0,C 180,E1 25908.677,E2 25908.677} C_VEL
LIN {X 0,Y 180.118,Z 784.604,A -85,B 0,C 180,E1 25914.176,E2 25914.176} C_VEL
LIN {X 0,Y 194.413,Z 772.398,A -85,B 0,C 180,E1 25916.11,E2 25916.11} C_VEL
LIN {X 0,Y 195.515,Z 770.629,A -85,B 0,C 180,E1 25920.005,E2 25920.005} C_VEL
LIN {X 0,Y 192.53,Z 773.718,A -85,B 0,C 180,E1 25926.756,E2 25926.756} C_VEL
LIN {X 0,Y 199.902,Z 790.728,A -85,B 0,C 180,E1 25954.485,E2 25954.485} C_VEL
LIN {X 0,Y 209.177,Z 798.489,A -85,B 0,C 180,E1 25963.832,E2 25963.832} C_VEL
LIN {X 0,Y 216.685,Z 805.196,A -85,B 0,C 180,E1 25971.19,E2 25971.19} C_VEL
LIN {X 0,Y 223.571,Z 811.477,A -85,B 0,C 180,E1 25979.31,E2 25979.31} C_VEL
LIN {X 0,Y 228.509,Z 816.02,A -85,B 0,C 180,E1 25986.66,E2 25986.66} C_VEL
LIN {X 0,Y 232.727,Z 819.635,A -85,B 0,C 180,E1 25994.97,E2 25994.97} C_VEL
LIN {X 0,Y 236.07,Z 821.157,A -85,B 0,C 180,E1 26002.657,E2 26002.657} C_VEL
LIN {X 0,Y 237.479,Z 821.489,A -85,B 0,C 180,E1 26010.002,E2 26010.002} C_VEL
LIN {X 0,Y 235.987,Z 821.139,A -85,B 0,C 180,E1 26017.349,E2 26017.349} C_VEL
LIN {X 0,Y 232.739,Z 819.652,A -85,B 0,C 180,E1 26025.033,E2 26025.033} C_VEL
LIN {X 0,Y 228.484,Z 815.957,A -85,B 0,C 180,E1 26033.347,E2 26033.347} C_VEL
LIN {X 0,Y 223.482,Z 811.497,A -85,B 0,C 180,E1 26040.679,E2 26040.679} C_VEL
LIN {X 0,Y 216.578,Z 805.164,A -85,B 0,C 180,E1 26048.837,E2 26048.837} C_VEL
LIN {X 0,Y 208.401,Z 797.735,A -85,B 0,C 180,E1 26056.942,E2 26056.942} C_VEL
LIN {X 0,Y 197.62,Z 789.054,A -85,B 0,C 180,E1 26068.047,E2 26068.047} C_VEL
LIN {X 0,Y 190.781,Z 788.237,A -85,B 0,C 180,E1 26072.805,E2 26072.805} C_VEL
LIN {X 0,Y 185.038,Z 787.542,A -85,B 0,C 180,E1 26077.876,E2 26077.876} C_VEL
LIN {X 0,Y 187.263,Z 777.645,A -85,B 0,C 180,E1 26095.373,E2 26095.373} C_VEL
LIN {X 0,Y 189.434,Z 775.88,A -85,B 0,C 180,E1 26099.995,E2 26099.995} C_VEL
LIN {X 0,Y 188.873,Z 776.619,A -85,B 0,C 180,E1 26101.954,E2 26101.954} C_VEL
LIN {X 0,Y 181.346,Z 782.837,A -85,B 0,C 180,E1 26103.054,E2 26103.054} C_VEL
LIN {X 0,Y 148.409,Z 805.774,A -85,B 0,C 180,E1 26107.512,E2 26107.512} C_VEL
LIN {X 0,Y 113.761,Z 824.213,A -85,B 0,C 180,E1 26115.376,E2 26115.376} C_VEL
LIN {X 0,Y 85.268,Z 835.757,A -85,B 0,C 180,E1 26127.755,E2 26127.755} C_VEL
LIN {X 0,Y 61.92,Z 843.361,A -85,B 0,C 180,E1 26152.456,E2 26152.456} C_VEL
LIN {X 0,Y 55.342,Z 845.581,A -85,B 0,C 180,E1 26174.169,E2 26174.169} C_VEL
LIN {X 0,Y 54.812,Z 846.018,A -85,B 0,C 180,E1 26189.993,E2 26189.993} C_VEL
LIN {X 0,Y 59.005,Z 844.339,A -85,B 0,C 180,E1 26220.755,E2 26220.755} C_VEL
LIN {X 0,Y 79.703,Z 837.681,A -85,B 0,C 180,E1 26248.418,E2 26248.418} C_VEL
LIN {X 0,Y 110.183,Z 825.793,A -85,B 0,C 180,E1 26263.459,E2 26263.459} C_VEL
LIN {X 0,Y 144.799,Z 807.922,A -85,B 0,C 180,E1 26271.884,E2 26271.884} C_VEL
LIN {X 0,Y 179.476,Z 784.352,A -85,B 0,C 180,E1 26276.755,E2 26276.755} C_VEL
LIN {X 0,Y 188.86,Z 776.628,A -85,B 0,C 180,E1 26278.055,E2 26278.055} C_VEL
LIN {X 0,Y 189.418,Z 775.893,A -85,B 0,C 180,E1 26280.005,E2 26280.005} C_VEL
LIN {X 0,Y 185.136,Z 780.366,A -85,B 0,C 180,E1 26289.387,E2 26289.387} C_VEL
LIN {X 0,Y 193.13,Z 794.725,A -85,B 0,C 180,E1 26314.647,E2 26314.647} C_VEL
LIN {X 0,Y 202.042,Z 801.841,A -85,B 0,C 180,E1 26323.998,E2 26323.998} C_VEL
LIN {X 0,Y 210.196,Z 809.045,A -85,B 0,C 180,E1 26332.163,E2 26332.163} C_VEL
LIN {X 0,Y 217.51,Z 815.541,A -85,B 0,C 180,E1 26340.948,E2 26340.948} C_VEL
LIN {X 0,Y 222.212,Z 820.121,A -85,B 0,C 180,E1 26348.689,E2 26348.689} C_VEL
LIN {X 0,Y 225.061,Z 822.471,A -85,B 0,C 180,E1 26354.445,E2 26354.445} C_VEL
LIN {X 0,Y 228.679,Z 824.267,A -85,B 0,C 180,E1 26362.418,E2 26362.418} C_VEL
LIN {X 0,Y 230.189,Z 824.533,A -85,B 0,C 180,E1 26370.002,E2 26370.002} C_VEL
LIN {X 0,Y 228.581,Z 824.251,A -85,B 0,C 180,E1 26377.589,E2 26377.589} C_VEL
LIN {X 0,Y 225.104,Z 822.499,A -85,B 0,C 180,E1 26385.556,E2 26385.556} C_VEL
LIN {X 0,Y 222.181,Z 820.066,A -85,B 0,C 180,E1 26391.315,E2 26391.315} C_VEL
LIN {X 0,Y 217.451,Z 815.556,A -85,B 0,C 180,E1 26399.065,E2 26399.065} C_VEL
LIN {X 0,Y 210.111,Z 809.093,A -85,B 0,C 180,E1 26407.807,E2 26407.807} C_VEL
LIN {X 0,Y 202.055,Z 801.832,A -85,B 0,C 180,E1 26416.005,E2 26416.005} C_VEL
LIN {X 0,Y 191.971,Z 793.961,A -85,B 0,C 180,E1 26426.611,E2 26426.611} C_VEL
LIN {X 0,Y 185.038,Z 787.542,A -85,B 0,C 180,E1 26437.876,E2 26437.876} C_VEL
LIN {X 0,Y 180.772,Z 786.919,A -85,B 0,C 180,E1 26443.203,E2 26443.203} C_VEL
LIN {X 0,Y 178.145,Z 786.236,A -85,B 0,C 180,E1 26448.733,E2 26448.733} C_VEL
LIN {X 0,Y 183.136,Z 780.915,A -85,B 0,C 180,E1 26459.995,E2 26459.995} C_VEL
LIN {X 0,Y 167.968,Z 792.345,A -85,B 0,C 180,E1 26461.808,E2 26461.808} C_VEL
LIN {X 0,Y 134.706,Z 812.782,A -85,B 0,C 180,E1 26466.425,E2 26466.425} C_VEL
LIN {X 0,Y 97.941,Z 829.712,A -85,B 0,C 180,E1 26475.629,E2 26475.629} C_VEL
LIN {X 0,Y 65.43,Z 840.467,A -85,B 0,C 180,E1 26494.56,E2 26494.56} C_VEL
LIN {X 0,Y 52.241,Z 844.089,A -85,B 0,C 180,E1 26514.701,E2 26514.701} C_VEL
LIN {X 0,Y 46.873,Z 845.771,A -85,B 0,C 180,E1 26549.991,E2 26549.991} C_VEL
LIN {X 0,Y 52.251,Z 844.091,A -85,B 0,C 180,E1 26585.273,E2 26585.273} C_VEL
LIN {X 0,Y 75.751,Z 837.43,A -85,B 0,C 180,E1 26613.68,E2 26613.68} C_VEL
LIN {X 0,Y 108.14,Z 825.537,A -85,B 0,C 180,E1 26627.615,E2 26627.615} C_VEL
LIN {X 0,Y 143.875,Z 807.672,A -85,B 0,C 180,E1 26635.1,E2 26635.1} C_VEL
LIN {X 0,Y 179.2,Z 784.101,A -85,B 0,C 180,E1 26639.336,E2 26639.336} C_VEL
LIN {X 0,Y 183.122,Z 780.925,A -85,B 0,C 180,E1 26640.005,E2 26640.005} C_VEL
LIN {X 0,Y 178.607,Z 785.408,A -85,B 0,C 180,E1 26649.733,E2 26649.733} C_VEL
LIN {X 0,Y 186.031,Z 798.366,A -85,B 0,C 180,E1 26674.603,E2 26674.603} C_VEL
LIN {X 0,Y 194.848,Z 805.057,A -85,B 0,C 180,E1 26684.193,E2 26684.193} C_VEL
LIN {X 0,Y 202.816,Z 811.922,A -85,B 0,C 180,E1 26692.293,E2 26692.293} C_VEL
LIN {X 0,Y 209.251,Z 817.661,A -85,B 0,C 180,E1 26699.933,E2 26699.933} C_VEL
LIN {X 0,Y 213.682,Z 821.756,A -85,B 0,C 180,E1 26706.652,E2 26706.652} C_VEL
LIN {X 0,Y 218.134,Z 825.65,A -85,B 0,C 180,E1 26715.593,E2 26715.593} C_VEL
LIN {X 0,Y 221.119,Z 826.973,A -85,B 0,C 180,E1 26722.157,E2 26722.157} C_VEL
LIN {X 0,Y 222.25,Z 827.295,A -85,B 0,C 180,E1 26726.109,E2 26726.109} C_VEL
LIN {X 0,Y 222.806,Z 827.33,A -85,B 0,C 180,E1 26730.002,E2 26730.002} C_VEL
LIN {X 0,Y 222.204,Z 827.28,A -85,B 0,C 180,E1 26733.896,E2 26733.896} C_VEL
LIN {X 0,Y 219.362,Z 826.3,A -85,B 0,C 180,E1 26741.912,E2 26741.912} C_VEL
LIN {X 0,Y 215.135,Z 823.192,A -85,B 0,C 180,E1 26750.533,E2 26750.533} C_VEL
LIN {X 0,Y 210.957,Z 819.184,A -85,B 0,C 180,E1 26757.654,E2 26757.654} C_VEL
LIN {X 0,Y 203.895,Z 813.121,A -85,B 0,C 180,E1 26766.307,E2 26766.307} C_VEL
LIN {X 0,Y 197.016,Z 806.943,A -85,B 0,C 180,E1 26773.581,E2 26773.581} C_VEL
LIN {X 0,Y 187.462,Z 799.533,A -85,B 0,C 180,E1 26783.611,E2 26783.611} C_VEL
LIN {X 0,Y 177.522,Z 788.124,A -85,B 0,C 180,E1 26805.221,E2 26805.221} C_VEL
LIN {X 0,Y 178.145,Z 786.236,A -85,B 0,C 180,E1 26808.733,E2 26808.733} C_VEL
LIN {X 0,Y 176.257,Z 786.579,A -85,B 0,C 180,E1 26812.492,E2 26812.492} C_VEL
LIN {X 0,Y 174.846,Z 787.137,A -85,B 0,C 180,E1 26816.346,E2 26816.346} C_VEL
LIN {X 0,Y 175.627,Z 786.538,A -85,B 0,C 180,E1 26817.904,E2 26817.904} C_VEL
LIN {X 0,Y 169.805,Z 790.739,A -85,B 0,C 180,E1 26818.841,E2 26818.841} C_VEL
LIN {X 0,Y 135.967,Z 811.552,A -85,B 0,C 180,E1 26822.688,E2 26822.688} C_VEL
LIN {X 0,Y 99.411,Z 828.169,A -85,B 0,C 180,E1 26829.949,E2 26829.949} C_VEL
LIN {X 0,Y 66.277,Z 838.935,A -85,B 0,C 180,E1 26844.379,E2 26844.379} C_VEL
LIN {X 0,Y 45.886,Z 843.839,A -85,B 0,C 180,E1 26868.862,E2 26868.862} C_VEL
LIN {X 0,Y 38.944,Z 845.525,A -85,B 0,C 180,E1 26909.99,E2 26909.99} C_VEL
LIN {X 0,Y 45.895,Z 843.841,A -85,B 0,C 180,E1 26951.105,E2 26951.105} C_VEL
LIN {X 0,Y 72.502,Z 837.179,A -85,B 0,C 180,E1 26979.472,E2 26979.472} C_VEL
LIN {X 0,Y 110.278,Z 823.822,A -85,B 0,C 180,E1 26992.75,E2 26992.75} C_VEL
LIN {X 0,Y 149.029,Z 804.208,A -85,B 0,C 180,E1 26999.033,E2 26999.033} C_VEL
LIN {X 0,Y 173.347,Z 788.211,A -85,B 0,C 180,E1 27001.465,E2 27001.465} C_VEL
LIN {X 0,Y 175.628,Z 786.537,A -85,B 0,C 180,E1 27002.104,E2 27002.104} C_VEL
LIN {X 0,Y 177.978,Z 801.391,A -85,B 0,C 180,E1 27033.446,E2 27033.446} C_VEL
LIN {X 0,Y 186.517,Z 807.411,A -85,B 0,C 180,E1 27043.272,E2 27043.272} C_VEL
LIN {X 0,Y 194.544,Z 813.833,A -85,B 0,C 180,E1 27051.648,E2 27051.648} C_VEL
LIN {X 0,Y 200.112,Z 818.908,A -85,B 0,C 180,E1 27058.142,E2 27058.142} C_VEL
LIN {X 0,Y 205.604,Z 823.678,A -85,B 0,C 180,E1 27065.676,E2 27065.676} C_VEL
LIN {X 0,Y 209.423,Z 827.308,A -85,B 0,C 180,E1 27073.25,E2 27073.25} C_VEL
LIN {X 0,Y 213.439,Z 829.457,A -85,B 0,C 180,E1 27081.873,E2 27081.873} C_VEL
LIN {X 0,Y 214.712,Z 829.858,A -85,B 0,C 180,E1 27085.972,E2 27085.972} C_VEL
LIN {X 0,Y 215.347,Z 829.915,A -85,B 0,C 180,E1 27090.002,E2 27090.002} C_VEL
LIN {X 0,Y 214.661,Z 829.842,A -85,B 0,C 180,E1 27094.033,E2 27094.033} C_VEL
LIN {X 0,Y 211.577,Z 828.62,A -85,B 0,C 180,E1 27102.357,E2 27102.357} C_VEL
LIN {X 0,Y 208.059,Z 826.168,A -85,B 0,C 180,E1 27109.452,E2 27109.452} C_VEL
LIN {X 0,Y 203.674,Z 821.955,A -85,B 0,C 180,E1 27117.235,E2 27117.235} C_VEL
LIN {X 0,Y 197.412,Z 816.647,A -85,B 0,C 180,E1 27124.93,E2 27124.93} C_VEL
LIN {X 0,Y 191.25,Z 811.097,A -85,B 0,C 180,E1 27131.734,E2 27131.734} C_VEL
LIN {X 0,Y 184.265,Z 805.802,A -85,B 0,C 180,E1 27139.064,E2 27139.064} C_VEL
LIN {X 0,Y 175.157,Z 799.461,A -85,B 0,C 180,E1 27150.403,E2 27150.403} C_VEL
LIN {X 0,Y 174.846,Z 787.137,A -85,B 0,C 180,E1 27176.346,E2 27176.346} C_VEL
LIN {X 0,Y 172.576,Z 788.751,A -85,B 0,C 180,E1 27177.352,E2 27177.352} C_VEL
LIN {X 0,Y 164.881,Z 794.096,A -85,B 0,C 180,E1 27177.42,E2 27177.42} C_VEL
LIN {X 0,Y 155.278,Z 800.236,A -85,B 0,C 180,E1 27177.28,E2 27177.28} C_VEL
LIN {X 0,Y 120.752,Z 818.648,A -85,B 0,C 180,E1 27181.156,E2 27181.156} C_VEL
LIN {X 0,Y 84.028,Z 832.83,A -85,B 0,C 180,E1 27188.994,E2 27188.994} C_VEL
LIN {X 0,Y 50.778,Z 841.539,A -85,B 0,C 180,E1 27206.916,E2 27206.916} C_VEL
LIN {X 0,Y 32.896,Z 844.836,A -85,B 0,C 180,E1 27242.681,E2 27242.681} C_VEL
LIN {X 0,Y 30.998,Z 845.278,A -85,B 0,C 180,E1 27269.987,E2 27269.987} C_VEL
LIN {X 0,Y 40.157,Z 843.592,A -85,B 0,C 180,E1 27318.71,E2 27318.71} C_VEL
LIN {X 0,Y 70.056,Z 836.928,A -85,B 0,C 180,E1 27345.742,E2 27345.742} C_VEL
LIN {X 0,Y 109.544,Z 823.565,A -85,B 0,C 180,E1 27357.019,E2 27357.019} C_VEL
LIN {X 0,Y 149.113,Z 803.958,A -85,B 0,C 180,E1 27362.154,E2 27362.154} C_VEL
LIN {X 0,Y 168.105,Z 791.952,A -85,B 0,C 180,E1 27364,E2 27364} C_VEL
LIN {X 0,Y 171.8,Z 805.506,A -85,B 0,C 180,E1 27394.821,E2 27394.821} C_VEL
LIN {X 0,Y 180.608,Z 811.433,A -85,B 0,C 180,E1 27405.064,E2 27405.064} C_VEL
LIN {X 0,Y 188.297,Z 817.389,A -85,B 0,C 180,E1 27413.271,E2 27413.271} C_VEL
LIN {X 0,Y 195.099,Z 823.293,A -85,B 0,C 180,E1 27421.434,E2 27421.434} C_VEL
LIN {X 0,Y 198.967,Z 826.962,A -85,B 0,C 180,E1 27427.717,E2 27427.717} C_VEL
LIN {X 0,Y 203.658,Z 830.679,A -85,B 0,C 180,E1 27437.159,E2 27437.159} C_VEL
LIN {X 0,Y 205.64,Z 831.688,A -85,B 0,C 180,E1 27441.563,E2 27441.563} C_VEL
LIN {X 0,Y 207.023,Z 832.055,A -85,B 0,C 180,E1 27445.822,E2 27445.822} C_VEL
LIN {X 0,Y 207.735,Z 832.088,A -85,B 0,C 180,E1 27450.002,E2 27450.002} C_VEL
LIN {X 0,Y 206.975,Z 832.034,A -85,B 0,C 180,E1 27454.183,E2 27454.183} C_VEL
LIN {X 0,Y 205.547,Z 831.654,A -85,B 0,C 180,E1 27458.445,E2 27458.445} C_VEL
LIN {X 0,Y 202.721,Z 830.155,A -85,B 0,C 180,E1 27464.59,E2 27464.59} C_VEL
LIN {X 0,Y 198.93,Z 826.918,A -85,B 0,C 180,E1 27472.291,E2 27472.291} C_VEL
LIN {X 0,Y 195.021,Z 823.284,A -85,B 0,C 180,E1 27478.552,E2 27478.552} C_VEL
LIN {X 0,Y 188.22,Z 817.445,A -85,B 0,C 180,E1 27486.698,E2 27486.698} C_VEL
LIN {X 0,Y 180.595,Z 811.423,A -85,B 0,C 180,E1 27494.951,E2 27494.951} C_VEL
LIN {X 0,Y 171.754,Z 805.537,A -85,B 0,C 180,E1 27505.168,E2 27505.168} C_VEL
LIN {X 0,Y 168.121,Z 791.94,A -85,B 0,C 180,E1 27536.018,E2 27536.018} C_VEL
LIN {X 0,Y 155.278,Z 800.236,A -85,B 0,C 180,E1 27537.28,E2 27537.28} C_VEL
LIN {X 0,Y 140.049,Z 808.981,A -85,B 0,C 180,E1 27537.095,E2 27537.095} C_VEL
LIN {X 0,Y 124.385,Z 816.814,A -85,B 0,C 180,E1 27536.914,E2 27536.914} C_VEL
LIN {X 0,Y 83.152,Z 832.578,A -85,B 0,C 180,E1 27543.437,E2 27543.437} C_VEL
LIN {X 0,Y 46.888,Z 841.414,A -85,B 0,C 180,E1 27558.753,E2 27558.753} C_VEL
LIN {X 0,Y 26.025,Z 844.587,A -85,B 0,C 180,E1 27594.542,E2 27594.542} C_VEL
LIN {X 0,Y 23.07,Z 845.032,A -85,B 0,C 180,E1 27629.982,E2 27629.982} C_VEL
LIN {X 0,Y 35.346,Z 843.342,A -85,B 0,C 180,E1 27688.611,E2 27688.611} C_VEL
LIN {X 0,Y 68.275,Z 836.739,A -85,B 0,C 180,E1 27712.291,E2 27712.291} C_VEL
LIN {X 0,Y 109.424,Z 823.31,A -85,B 0,C 180,E1 27721.301,E2 27721.301} C_VEL
LIN {X 0,Y 149.638,Z 803.709,A -85,B 0,C 180,E1 27725.262,E2 27725.262} C_VEL
LIN {X 0,Y 156.851,Z 799.39,A -85,B 0,C 180,E1 27725.736,E2 27725.736} C_VEL
LIN {X 0,Y 160.022,Z 797.457,A -85,B 0,C 180,E1 27726.425,E2 27726.425} C_VEL
LIN {X 0,Y 165.62,Z 809.487,A -85,B 0,C 180,E1 27756.318,E2 27756.318} C_VEL
LIN {X 0,Y 175.32,Z 815.685,A -85,B 0,C 180,E1 27767.659,E2 27767.659} C_VEL
LIN {X 0,Y 182.6,Z 821.168,A -85,B 0,C 180,E1 27775.738,E2 27775.738} C_VEL
LIN {X 0,Y 187.798,Z 825.562,A -85,B 0,C 180,E1 27782.123,E2 27782.123} C_VEL
LIN {X 0,Y 192.513,Z 830.062,A -85,B 0,C 180,E1 27790.167,E2 27790.167} C_VEL
LIN {X 0,Y 195.64,Z 832.456,A -85,B 0,C 180,E1 27796.623,E2 27796.623} C_VEL
LIN {X 0,Y 198.06,Z 833.577,A -85,B 0,C 180,E1 27802.109,E2 27802.109} C_VEL
LIN {X 0,Y 200.063,Z 834.026,A -85,B 0,C 180,E1 27810.002,E2 27810.002} C_VEL
LIN {X 0,Y 198.006,Z 833.583,A -85,B 0,C 180,E1 27817.779,E2 27817.779} C_VEL
LIN {X 0,Y 195.639,Z 832.5,A -85,B 0,C 180,E1 27823.381,E2 27823.381} C_VEL
LIN {X 0,Y 192.487,Z 830.042,A -85,B 0,C 180,E1 27829.812,E2 27829.812} C_VEL
LIN {X 0,Y 187.756,Z 825.6,A -85,B 0,C 180,E1 27837.853,E2 27837.853} C_VEL
LIN {X 0,Y 179.963,Z 819.14,A -85,B 0,C 180,E1 27847.193,E2 27847.193} C_VEL
LIN {X 0,Y 172.435,Z 813.787,A -85,B 0,C 180,E1 27855.559,E2 27855.559} C_VEL
LIN {X 0,Y 163.582,Z 808.35,A -85,B 0,C 180,E1 27866.387,E2 27866.387} C_VEL
LIN {X 0,Y 160.036,Z 797.448,A -85,B 0,C 180,E1 27893.576,E2 27893.576} C_VEL
LIN {X 0,Y 156.673,Z 799.504,A -85,B 0,C 180,E1 27894.243,E2 27894.243} C_VEL
LIN {X 0,Y 124.385,Z 816.814,A -85,B 0,C 180,E1 27896.914,E2 27896.914} C_VEL
LIN {X 0,Y 108.264,Z 823.693,A -85,B 0,C 180,E1 27896.736,E2 27896.736} C_VEL
LIN {X 0,Y 91.76,Z 829.599,A -85,B 0,C 180,E1 27896.504,E2 27896.504} C_VEL
LIN {X 0,Y 53.045,Z 839.676,A -85,B 0,C 180,E1 27905.251,E2 27905.251} C_VEL
LIN {X 0,Y 20.039,Z 844.339,A -85,B 0,C 180,E1 27941.116,E2 27941.116} C_VEL
LIN {X 0,Y 15.078,Z 844.781,A -85,B 0,C 180,E1 27991.277,E2 27991.277} C_VEL
LIN {X 0,Y 31.892,Z 843.092,A -85,B 0,C 180,E1 28061.102,E2 28061.102} C_VEL
LIN {X 0,Y 71.376,Z 835.542,A -85,B 0,C 180,E1 28080.013,E2 28080.013} C_VEL
LIN {X 0,Y 109.915,Z 823.054,A -85,B 0,C 180,E1 28085.571,E2 28085.571} C_VEL
LIN {X 0,Y 150.685,Z 803.411,A -85,B 0,C 180,E1 28088.339,E2 28088.339} C_VEL
LIN {X 0,Y 152.19,Z 802.555,A -85,B 0,C 180,E1 28088.559,E2 28088.559} C_VEL
LIN {X 0,Y 157.354,Z 812.044,A -85,B 0,C 180,E1 28115.134,E2 28115.134} C_VEL
LIN {X 0,Y 166.537,Z 817.419,A -85,B 0,C 180,E1 28126.466,E2 28126.466} C_VEL
LIN {X 0,Y 173.622,Z 822.142,A -85,B 0,C 180,E1 28134.418,E2 28134.418} C_VEL
LIN {X 0,Y 180.708,Z 827.852,A -85,B 0,C 180,E1 28143.296,E2 28143.296} C_VEL
LIN {X 0,Y 185.082,Z 831.928,A -85,B 0,C 180,E1 28150.968,E2 28150.968} C_VEL
LIN {X 0,Y 189.678,Z 835.038,A -85,B 0,C 180,E1 28160.847,E2 28160.847} C_VEL
LIN {X 0,Y 191.422,Z 835.627,A -85,B 0,C 180,E1 28165.481,E2 28165.481} C_VEL
LIN {X 0,Y 192.347,Z 835.729,A -85,B 0,C 180,E1 28170.002,E2 28170.002} C_VEL
LIN {X 0,Y 191.37,Z 835.599,A -85,B 0,C 180,E1 28174.525,E2 28174.525} C_VEL
LIN {X 0,Y 189.606,Z 835.02,A -85,B 0,C 180,E1 28179.161,E2 28179.161} C_VEL
LIN {X 0,Y 187.113,Z 833.671,A -85,B 0,C 180,E1 28184.571,E2 28184.571} C_VEL
LIN {X 0,Y 184.125,Z 831.152,A -85,B 0,C 180,E1 28190.752,E2 28190.752} C_VEL
LIN {X 0,Y 180.657,Z 827.865,A -85,B 0,C 180,E1 28196.694,E2 28196.694} C_VEL
LIN {X 0,Y 173.52,Z 822.161,A -85,B 0,C 180,E1 28205.588,E2 28205.588} C_VEL
LIN {X 0,Y 166.542,Z 817.417,A -85,B 0,C 180,E1 28213.535,E2 28213.535} C_VEL
LIN {X 0,Y 157.272,Z 812.093,A -85,B 0,C 180,E1 28224.845,E2 28224.845} C_VEL
LIN {X 0,Y 152.203,Z 802.547,A -85,B 0,C 180,E1 28251.442,E2 28251.442} C_VEL
LIN {X 0,Y 113.792,Z 821.441,A -85,B 0,C 180,E1 28254.067,E2 28254.067} C_VEL
LIN {X 0,Y 91.76,Z 829.599,A -85,B 0,C 180,E1 28256.504,E2 28256.504} C_VEL
LIN {X 0,Y 74.942,Z 834.552,A -85,B 0,C 180,E1 28256.153,E2 28256.153} C_VEL
LIN {X 0,Y 57.838,Z 838.466,A -85,B 0,C 180,E1 28255.48,E2 28255.48} C_VEL
LIN {X 0,Y 30.266,Z 842.838,A -85,B 0,C 180,E1 28264.132,E2 28264.132} C_VEL
LIN {X 0,Y 7.182,Z 844.538,A -85,B 0,C 180,E1 28349.944,E2 28349.944} C_VEL
LIN {X 0,Y 30.255,Z 842.841,A -85,B 0,C 180,E1 28435.792,E2 28435.792} C_VEL
LIN {X 0,Y 70.823,Z 835.544,A -85,B 0,C 180,E1 28446.431,E2 28446.431} C_VEL
LIN {X 0,Y 111.008,Z 822.799,A -85,B 0,C 180,E1 28449.775,E2 28449.775} C_VEL
LIN {X 0,Y 144.242,Z 807.489,A -85,B 0,C 180,E1 28451.446,E2 28451.446} C_VEL
LIN {X 0,Y 151.168,Z 815.749,A -85,B 0,C 180,E1 28477.009,E2 28477.009} C_VEL
LIN {X 0,Y 160.955,Z 821.021,A -85,B 0,C 180,E1 28488.987,E2 28488.987} C_VEL
LIN {X 0,Y 168.185,Z 825.681,A -85,B 0,C 180,E1 28497.432,E2 28497.432} C_VEL
LIN {X 0,Y 173.397,Z 829.643,A -85,B 0,C 180,E1 28504.209,E2 28504.209} C_VEL
LIN {X 0,Y 177.931,Z 833.937,A -85,B 0,C 180,E1 28512.735,E2 28512.735} C_VEL
LIN {X 0,Y 182.481,Z 836.651,A -85,B 0,C 180,E1 28522.931,E2 28522.931} C_VEL
LIN {X 0,Y 184.548,Z 837.068,A -85,B 0,C 180,E1 28530.002,E2 28530.002} C_VEL
LIN {X 0,Y 182.464,Z 836.689,A -85,B 0,C 180,E1 28537.025,E2 28537.025} C_VEL
LIN {X 0,Y 177.901,Z 833.924,A -85,B 0,C 180,E1 28547.273,E2 28547.273} C_VEL
LIN {X 0,Y 173.325,Z 829.643,A -85,B 0,C 180,E1 28555.808,E2 28555.808} C_VEL
LIN {X 0,Y 166.028,Z 824.256,A -85,B 0,C 180,E1 28565.107,E2 28565.107} C_VEL
LIN {X 0,Y 158.085,Z 819.489,A -85,B 0,C 180,E1 28574.274,E2 28574.274} C_VEL
LIN {X 0,Y 148.962,Z 814.704,A -85,B 0,C 180,E1 28586.134,E2 28586.134} C_VEL
LIN {X 0,Y 144.247,Z 807.485,A -85,B 0,C 180,E1 28608.564,E2 28608.564} C_VEL
LIN {X 0,Y 107.127,Z 824.252,A -85,B 0,C 180,E1 28610.436,E2 28610.436} C_VEL
LIN {X 0,Y 65.67,Z 836.784,A -85,B 0,C 180,E1 28614.263,E2 28614.263} C_VEL
LIN {X 0,Y 57.838,Z 838.466,A -85,B 0,C 180,E1 28615.48,E2 28615.48} C_VEL
LIN {X 0,Y 40.612,Z 841.359,A -85,B 0,C 180,E1 28613.941,E2 28613.941} C_VEL
LIN {X 0,Y 23.309,Z 843.194,A -85,B 0,C 180,E1 28608.945,E2 28608.945} C_VEL
LIN {X 0,Y 0.786,Z 844.291,A -85,B 0,C 180,E1 28530.515,E2 28530.515} C_VEL
LIN {X 0,Y 30.743,Z 842.589,A -85,B 0,C 180,E1 28451.046,E2 28451.046} C_VEL
LIN {X 0,Y 72.409,Z 835.241,A -85,B 0,C 180,E1 28452.894,E2 28452.894} C_VEL
LIN {X 0,Y 112.65,Z 822.557,A -85,B 0,C 180,E1 28453.879,E2 28453.879} C_VEL
LIN {X 0,Y 136.573,Z 812.083,A -85,B 0,C 180,E1 28454.591,E2 28454.591} C_VEL
LIN {X 0,Y 144.782,Z 819.102,A -85,B 0,C 180,E1 28478.716,E2 28478.716} C_VEL
LIN {X 0,Y 154.95,Z 824.196,A -85,B 0,C 180,E1 28491.186,E2 28491.186} C_VEL
LIN {X 0,Y 162.118,Z 828.496,A -85,B 0,C 180,E1 28499.833,E2 28499.833} C_VEL
LIN {X 0,Y 166.081,Z 831.373,A -85,B 0,C 180,E1 28505.323,E2 28505.323} C_VEL
LIN {X 0,Y 170.921,Z 835.577,A -85,B 0,C 180,E1 28514.644,E2 28514.644} C_VEL
LIN {X 0,Y 173.326,Z 837.12,A -85,B 0,C 180,E1 28519.975,E2 28519.975} C_VEL
LIN {X 0,Y 175.475,Z 837.938,A -85,B 0,C 180,E1 28525.069,E2 28525.069} C_VEL
LIN {X 0,Y 176.667,Z 838.109,A -85,B 0,C 180,E1 28530.002,E2 28530.002} C_VEL
LIN {X 0,Y 175.409,Z 837.903,A -85,B 0,C 180,E1 28534.937,E2 28534.937} C_VEL
LIN {X 0,Y 171.383,Z 835.955,A -85,B 0,C 180,E1 28544.392,E2 28544.392} C_VEL
LIN {X 0,Y 168.074,Z 833.185,A -85,B 0,C 180,E1 28551.049,E2 28551.049} C_VEL
LIN {X 0,Y 164.128,Z 829.965,A -85,B 0,C 180,E1 28557.371,E2 28557.371} C_VEL
LIN {X 0,Y 158.21,Z 826.052,A -85,B 0,C 180,E1 28564.913,E2 28564.913} C_VEL
LIN {X 0,Y 149.569,Z 821.418,A -85,B 0,C 180,E1 28575.063,E2 28575.063} C_VEL
LIN {X 0,Y 139.305,Z 816.411,A -85,B 0,C 180,E1 28590.071,E2 28590.071} C_VEL
LIN {X 0,Y 136.56,Z 812.082,A -85,B 0,C 180,E1 28605.441,E2 28605.441} C_VEL
LIN {X 0,Y 103.925,Z 825.777,A -85,B 0,C 180,E1 28606.272,E2 28606.272} C_VEL
LIN {X 0,Y 61.842,Z 837.675,A -85,B 0,C 180,E1 28607.462,E2 28607.462} C_VEL
LIN {X 0,Y 23.309,Z 843.194,A -85,B 0,C 180,E1 28608.945,E2 28608.945} C_VEL
LIN {X 0,Y 10.925,Z 843.961,A -85,B 0,C 180,E1 28593.123,E2 28593.123} C_VEL
LIN {X 0,Y 16.056,Z 843.679,A -85,B 0,C 180,E1 28480.944,E2 28480.944} C_VEL
LIN {X 0,Y 48.567,Z 840.286,A -85,B 0,C 180,E1 28461.256,E2 28461.256} C_VEL
LIN {X 0,Y 91.416,Z 830.398,A -85,B 0,C 180,E1 28458.362,E2 28458.362} C_VEL
LIN {X 0,Y 129.249,Z 816.356,A -85,B 0,C 180,E1 28457.891,E2 28457.891} C_VEL
LIN {X 0,Y 138.546,Z 822.275,A -85,B 0,C 180,E1 28480.814,E2 28480.814} C_VEL
LIN {X 0,Y 147.85,Z 826.459,A -85,B 0,C 180,E1 28492.242,E2 28492.242} C_VEL
LIN {X 0,Y 155.07,Z 830.449,A -85,B 0,C 180,E1 28501.151,E2 28501.151} C_VEL
LIN {X 0,Y 160.64,Z 834.435,A -85,B 0,C 180,E1 28509.961,E2 28509.961} C_VEL
LIN {X 0,Y 165.084,Z 837.673,A -85,B 0,C 180,E1 28519.469,E2 28519.469} C_VEL
LIN {X 0,Y 167.371,Z 838.624,A -85,B 0,C 180,E1 28524.83,E2 28524.83} C_VEL
LIN {X 0,Y 168.759,Z 838.843,A -85,B 0,C 180,E1 28530.002,E2 28530.002} C_VEL
LIN {X 0,Y 166.908,Z 838.522,A -85,B 0,C 180,E1 28535.966,E2 28535.966} C_VEL
LIN {X 0,Y 165.049,Z 837.686,A -85,B 0,C 180,E1 28540.539,E2 28540.539} C_VEL
LIN {X 0,Y 160.614,Z 834.448,A -85,B 0,C 180,E1 28550.014,E2 28550.014} C_VEL
LIN {X 0,Y 154.702,Z 830.3,A -85,B 0,C 180,E1 28559.193,E2 28559.193} C_VEL
LIN {X 0,Y 147.841,Z 826.455,A -85,B 0,C 180,E1 28567.768,E2 28567.768} C_VEL
LIN {X 0,Y 137.878,Z 822.041,A -85,B 0,C 180,E1 28580.011,E2 28580.011} C_VEL
LIN {X 0,Y 129.216,Z 816.362,A -85,B 0,C 180,E1 28602.144,E2 28602.144} C_VEL
LIN {X 0,Y 87.517,Z 831.572,A -85,B 0,C 180,E1 28601.516,E2 28601.516} C_VEL
LIN {X 0,Y 48.603,Z 840.282,A -85,B 0,C 180,E1 28598.683,E2 28598.683} C_VEL
LIN {X 0,Y 18.66,Z 843.589,A -85,B 0,C 180,E1 28584.006,E2 28584.006} C_VEL
LIN {X 0,Y 8.76,Z 844.043,A -85,B 0,C 180,E1 28530.046,E2 28530.046} C_VEL
LIN {X 0,Y 16.056,Z 843.679,A -85,B 0,C 180,E1 28480.944,E2 28480.944} C_VEL
LIN {X 0,Y 28.718,Z 842.846,A -85,B 0,C 180,E1 28472.131,E2 28472.131} C_VEL
LIN {X 0,Y 48.521,Z 840.549,A -85,B 0,C 180,E1 28470.729,E2 28470.729} C_VEL
LIN {X 0,Y 50.646,Z 840.236,A -85,B 0,C 180,E1 28470.104,E2 28470.104} C_VEL
LIN {X 0,Y 90.428,Z 831.326,A -85,B 0,C 180,E1 28463.404,E2 28463.404} C_VEL
LIN {X 0,Y 122.197,Z 820.273,A -85,B 0,C 180,E1 28461.752,E2 28461.752} C_VEL
LIN {X 0,Y 132.414,Z 825.308,A -85,B 0,C 180,E1 28483.148,E2 28483.148} C_VEL
LIN {X 0,Y 141.876,Z 829.155,A -85,B 0,C 180,E1 28494.772,E2 28494.772} C_VEL
LIN {X 0,Y 147.888,Z 832.154,A -85,B 0,C 180,E1 28502.349,E2 28502.349} C_VEL
LIN {X 0,Y 151.962,Z 834.725,A -85,B 0,C 180,E1 28508.763,E2 28508.763} C_VEL
LIN {X 0,Y 156.724,Z 837.983,A -85,B 0,C 180,E1 28518.9,E2 28518.9} C_VEL
LIN {X 0,Y 159.253,Z 839.003,A -85,B 0,C 180,E1 28524.565,E2 28524.565} C_VEL
LIN {X 0,Y 160.801,Z 839.315,A -85,B 0,C 180,E1 28530.003,E2 28530.003} C_VEL
LIN {X 0,Y 159.18,Z 839.004,A -85,B 0,C 180,E1 28535.442,E2 28535.442} C_VEL
LIN {X 0,Y 155.405,Z 837.223,A -85,B 0,C 180,E1 28543.808,E2 28543.808} C_VEL
LIN {X 0,Y 150.4,Z 833.783,A -85,B 0,C 180,E1 28553.664,E2 28553.664} C_VEL
LIN {X 0,Y 144.941,Z 830.654,A -85,B 0,C 180,E1 28561.373,E2 28561.373} C_VEL
LIN {X 0,Y 136.601,Z 826.911,A -85,B 0,C 180,E1 28571.518,E2 28571.518} C_VEL
LIN {X 0,Y 125.658,Z 822.683,A -85,B 0,C 180,E1 28587.212,E2 28587.212} C_VEL
LIN {X 0,Y 122.154,Z 820.293,A -85,B 0,C 180,E1 28598.24,E2 28598.24} C_VEL
LIN {X 0,Y 82.688,Z 833.471,A -85,B 0,C 180,E1 28595.861,E2 28595.861} C_VEL
LIN {X 0,Y 41.786,Z 841.5,A -85,B 0,C 180,E1 28586.218,E2 28586.218} C_VEL
LIN {X 0,Y 16.737,Z 843.795,A -85,B 0,C 180,E1 28530.024,E2 28530.024} C_VEL
LIN {X 0,Y 41.944,Z 841.477,A -85,B 0,C 180,E1 28473.635,E2 28473.635} C_VEL
LIN {X 0,Y 50.646,Z 840.236,A -85,B 0,C 180,E1 28470.104,E2 28470.104} C_VEL
LIN {X 0,Y 59.226,Z 838.917,A -85,B 0,C 180,E1 28468.992,E2 28468.992} C_VEL
LIN {X 0,Y 82.978,Z 834.096,A -85,B 0,C 180,E1 28469.623,E2 28469.623} C_VEL
LIN {X 0,Y 85.068,Z 833.549,A -85,B 0,C 180,E1 28469.33,E2 28469.33} C_VEL
LIN {X 0,Y 111.989,Z 825.139,A -85,B 0,C 180,E1 28466.016,E2 28466.016} C_VEL
LIN {X 0,Y 115.669,Z 823.899,A -85,B 0,C 180,E1 28466.149,E2 28466.149} C_VEL
LIN {X 0,Y 126.355,Z 828.067,A -85,B 0,C 180,E1 28485.78,E2 28485.78} C_VEL
LIN {X 0,Y 134.698,Z 831.038,A -85,B 0,C 180,E1 28495.938,E2 28495.938} C_VEL
LIN {X 0,Y 141.387,Z 834.095,A -85,B 0,C 180,E1 28504.731,E2 28504.731} C_VEL
LIN {X 0,Y 145.437,Z 836.519,A -85,B 0,C 180,E1 28511.867,E2 28511.867} C_VEL
LIN {X 0,Y 148.378,Z 838.249,A -85,B 0,C 180,E1 28518.267,E2 28518.267} C_VEL
LIN {X 0,Y 151.453,Z 839.325,A -85,B 0,C 180,E1 28525.165,E2 28525.165} C_VEL
LIN {X 0,Y 152.812,Z 839.569,A -85,B 0,C 180,E1 28530.003,E2 28530.003} C_VEL
LIN {X 0,Y 150.984,Z 839.261,A -85,B 0,C 180,E1 28535.739,E2 28535.739} C_VEL
LIN {X 0,Y 148.341,Z 838.248,A -85,B 0,C 180,E1 28541.742,E2 28541.742} C_VEL
LIN {X 0,Y 144.519,Z 835.886,A -85,B 0,C 180,E1 28549.976,E2 28549.976} C_VEL
LIN {X 0,Y 138.372,Z 832.706,A -85,B 0,C 180,E1 28559.245,E2 28559.245} C_VEL
LIN {X 0,Y 132.135,Z 830.153,A -85,B 0,C 180,E1 28566.915,E2 28566.915} C_VEL
LIN {X 0,Y 124.453,Z 827.44,A -85,B 0,C 180,E1 28576.683,E2 28576.683} C_VEL
LIN {X 0,Y 115.585,Z 823.934,A -85,B 0,C 180,E1 28593.833,E2 28593.833} C_VEL
LIN {X 0,Y 92.244,Z 831.573,A -85,B 0,C 180,E1 28591.776,E2 28591.776} C_VEL
LIN {X 0,Y 56.608,Z 839.776,A -85,B 0,C 180,E1 28583.114,E2 28583.114} C_VEL
LIN {X 0,Y 31.015,Z 843.089,A -85,B 0,C 180,E1 28559.128,E2 28559.128} C_VEL
LIN {X 0,Y 24.723,Z 843.547,A -85,B 0,C 180,E1 28530.016,E2 28530.016} C_VEL
LIN {X 0,Y 42.687,Z 841.836,A -85,B 0,C 180,E1 28485.021,E2 28485.021} C_VEL
LIN {X 0,Y 78.777,Z 835.168,A -85,B 0,C 180,E1 28470.468,E2 28470.468} C_VEL
LIN {X 0,Y 85.068,Z 833.549,A -85,B 0,C 180,E1 28469.33,E2 28469.33} C_VEL
LIN {X 0,Y 96.418,Z 830.734,A -85,B 0,C 180,E1 28469.665,E2 28469.665} C_VEL
LIN {X 0,Y 107.902,Z 827.685,A -85,B 0,C 180,E1 28470.785,E2 28470.785} C_VEL
LIN {X 0,Y 109.64,Z 827.175,A -85,B 0,C 180,E1 28470.798,E2 28470.798} C_VEL
LIN {X 0,Y 120.533,Z 830.575,A -85,B 0,C 180,E1 28488.702,E2 28488.702} C_VEL
LIN {X 0,Y 126.825,Z 832.594,A -85,B 0,C 180,E1 28496.408,E2 28496.408} C_VEL
LIN {X 0,Y 133.321,Z 835.107,A -85,B 0,C 180,E1 28504.904,E2 28504.904} C_VEL
LIN {X 0,Y 136.878,Z 836.802,A -85,B 0,C 180,E1 28510.69,E2 28510.69} C_VEL
LIN {X 0,Y 139.879,Z 838.52,A -85,B 0,C 180,E1 28517.543,E2 28517.543} C_VEL
LIN {X 0,Y 142.765,Z 839.519,A -85,B 0,C 180,E1 28523.935,E2 28523.935} C_VEL
LIN {X 0,Y 144.824,Z 839.817,A -85,B 0,C 180,E1 28530.003,E2 28530.003} C_VEL
LIN {X 0,Y 142.72,Z 839.519,A -85,B 0,C 180,E1 28536.072,E2 28536.072} C_VEL
LIN {X 0,Y 139.492,Z 838.347,A -85,B 0,C 180,E1 28543.167,E2 28543.167} C_VEL
LIN {X 0,Y 136.825,Z 836.801,A -85,B 0,C 180,E1 28549.324,E2 28549.324} C_VEL
LIN {X 0,Y 131.596,Z 834.435,A -85,B 0,C 180,E1 28557.305,E2 28557.305} C_VEL
LIN {X 0,Y 126.803,Z 832.604,A -85,B 0,C 180,E1 28563.578,E2 28563.578} C_VEL
LIN {X 0,Y 120.501,Z 830.589,A -85,B 0,C 180,E1 28571.28,E2 28571.28} C_VEL
LIN {X 0,Y 109.543,Z 827.213,A -85,B 0,C 180,E1 28589.166,E2 28589.166} C_VEL
LIN {X 0,Y 73.077,Z 837.274,A -85,B 0,C 180,E1 28581.706,E2 28581.706} C_VEL
LIN {X 0,Y 48.822,Z 841.58,A -85,B 0,C 180,E1 28568.193,E2 28568.193} C_VEL
LIN {X 0,Y 32.705,Z 843.299,A -85,B 0,C 180,E1 28530.012,E2 28530.012} C_VEL
LIN {X 0,Y 48.779,Z 841.583,A -85,B 0,C 180,E1 28491.789,E2 28491.789} C_VEL
LIN {X 0,Y 87.371,Z 833.815,A -85,B 0,C 180,E1 28474.335,E2 28474.335} C_VEL
LIN {X 0,Y 107.902,Z 827.685,A -85,B 0,C 180,E1 28470.785,E2 28470.785} C_VEL
LIN {X 0,Y 111.236,Z 827.193,A -85,B 0,C 180,E1 28472.486,E2 28472.486} C_VEL
LIN {X 0,Y 112.076,Z 828.522,A -85,B 0,C 180,E1 28477.542,E2 28477.542} C_VEL
LIN {X 0,Y 111.448,Z 832.037,A -85,B 0,C 180,E1 28487.602,E2 28487.602} C_VEL
LIN {X 0,Y 112.275,Z 832.333,A -85,B 0,C 180,E1 28488.975,E2 28488.975} C_VEL
LIN {X 0,Y 121.466,Z 834.882,A -85,B 0,C 180,E1 28500.429,E2 28500.429} C_VEL
LIN {X 0,Y 127.697,Z 837.108,A -85,B 0,C 180,E1 28509.24,E2 28509.24} C_VEL
LIN {X 0,Y 131.406,Z 838.791,A -85,B 0,C 180,E1 28516.725,E2 28516.725} C_VEL
LIN {X 0,Y 134.442,Z 839.779,A -85,B 0,C 180,E1 28523.558,E2 28523.558} C_VEL
LIN {X 0,Y 136.785,Z 840.067,A -85,B 0,C 180,E1 28530.003,E2 28530.003} C_VEL
LIN {X 0,Y 134.398,Z 839.78,A -85,B 0,C 180,E1 28536.45,E2 28536.45} C_VEL
LIN {X 0,Y 131.366,Z 838.791,A -85,B 0,C 180,E1 28543.285,E2 28543.285} C_VEL
LIN {X 0,Y 127.625,Z 837.108,A -85,B 0,C 180,E1 28550.779,E2 28550.779} C_VEL
LIN {X 0,Y 121.194,Z 834.806,A -85,B 0,C 180,E1 28559.875,E2 28559.875} C_VEL
LIN {X 0,Y 114.811,Z 832.957,A -85,B 0,C 180,E1 28567.933,E2 28567.933} C_VEL
LIN {X 0,Y 105.242,Z 830.574,A -85,B 0,C 180,E1 28581.558,E2 28581.558} C_VEL
LIN {X 0,Y 102.245,Z 830.709,A -85,B 0,C 180,E1 28583.808,E2 28583.808} C_VEL
LIN {X 0,Y 67.659,Z 839.268,A -85,B 0,C 180,E1 28572.005,E2 28572.005} C_VEL
LIN {X 0,Y 45.794,Z 842.587,A -85,B 0,C 180,E1 28549.249,E2 28549.249} C_VEL
LIN {X 0,Y 40.705,Z 843.051,A -85,B 0,C 180,E1 28530.01,E2 28530.01} C_VEL
LIN {X 0,Y 55.393,Z 841.331,A -85,B 0,C 180,E1 28496.995,E2 28496.995} C_VEL
LIN {X 0,Y 88.195,Z 834.657,A -85,B 0,C 180,E1 28479.658,E2 28479.658} C_VEL
LIN {X 0,Y 102.292,Z 830.693,A -85,B 0,C 180,E1 28476.173,E2 28476.173} C_VEL
LIN {X 0,Y 105.453,Z 830.571,A -85,B 0,C 180,E1 28478.612,E2 28478.612} C_VEL
LIN {X 0,Y 112.275,Z 832.333,A -85,B 0,C 180,E1 28488.975,E2 28488.975} C_VEL
LIN {X 0,Y 114.546,Z 834.124,A -85,B 0,C 180,E1 28495.393,E2 28495.393} C_VEL
